LIN {X 0,Y 299.708,Z 457.98,A -85,B 0,C 180,E1 14084.743,E2 14084.743} C_VEL
LIN {X 0,Y 296.211,Z 453.711,A -85,B 0,C 180,E1 14082.616,E2 14082.616} C_VEL
LIN {X 0,Y 295.184,Z 452.077,A -85,B 0,C 180,E1 14081.599,E2 14081.599} C_VEL
LIN {X 0,Y 292.946,Z 448.012,A -85,B 0,C 180,E1 14078.654,E2 14078.654} C_VEL
LIN {X 0,Y 289.678,Z 442.411,A -85,B 0,C 180,E1 14073.523,E2 14073.523} C_VEL
LIN {X 0,Y 286.095,Z 436.55,A -85,B 0,C 180,E1 14064.796,E2 14064.796} C_VEL
LIN {X 0,Y 284.905,Z 435.389,A -85,B 0,C 180,E1 14059.25,E2 14059.25} C_VEL
LIN {X 0,Y 285.029,Z 435.504,A -85,B 0,C 180,E1 14053.387,E2 14053.387} C_VEL
LIN {X 0,Y 286.2,Z 436.707,A -85,B 0,C 180,E1 14048.438,E2 14048.438} C_VEL
LIN {X 0,Y 289.921,Z 442.675,A -85,B 0,C 180,E1 14039.803,E2 14039.803} C_VEL
LIN {X 0,Y 292.386,Z 447.018,A -85,B 0,C 180,E1 14035.882,E2 14035.882} C_VEL
LIN {X 0,Y 293.361,Z 448.287,A -85,B 0,C 180,E1 14034.721,E2 14034.721} C_VEL
LIN {X 0,Y 295.59,Z 452.337,A -85,B 0,C 180,E1 14031.833,E2 14031.833} C_VEL
LIN {X 0,Y 296.578,Z 453.696,A -85,B 0,C 180,E1 14030.884,E2 14030.884} C_VEL
LIN {X 0,Y 300.049,Z 458.18,A -85,B 0,C 180,E1 14028.662,E2 14028.662} C_VEL
LIN {X 0,Y 301.804,Z 460.211,A -85,B 0,C 180,E1 14027.662,E2 14027.662} C_VEL
LIN {X 0,Y 306.682,Z 466.167,A -85,B 0,C 180,E1 14025.124,E2 14025.124} C_VEL
LIN {X 0,Y 310.986,Z 471.496,A -85,B 0,C 180,E1 14023.085,E2 14023.085} C_VEL
LIN {X 0,Y 315.406,Z 477.154,A -85,B 0,C 180,E1 14021.135,E2 14021.135} C_VEL
LIN {X 0,Y 322.296,Z 486.098,A -85,B 0,C 180,E1 14018.384,E2 14018.384} C_VEL
LIN {X 0,Y 330.826,Z 498.047,A -85,B 0,C 180,E1 14015.303,E2 14015.303} C_VEL
LIN {X 0,Y 339.793,Z 511.207,A -85,B 0,C 180,E1 14012.39,E2 14012.39} C_VEL
LIN {X 0,Y 350.07,Z 527.48,A -85,B 0,C 180,E1 14009.372,E2 14009.372} C_VEL
LIN {X 0,Y 356.807,Z 539.249,A -85,B 0,C 180,E1 14007.536,E2 14007.536} C_VEL
LIN {X 0,Y 344.249,Z 751.792,A -85,B 0,C 180,E1 14003.107,E2 14003.107} C_VEL
LIN {X 0,Y 341.578,Z 773.987,A -85,B 0,C 180,E1 14002.425,E2 14002.425} C_VEL
LIN {X 0,Y 338.028,Z 795.147,A -85,B 0,C 180,E1 14001.526,E2 14001.526} C_VEL
LIN {X 0,Y 334.008,Z 814.782,A -85,B 0,C 180,E1 14000.432,E2 14000.432} C_VEL
LIN {X 0,Y 329.123,Z 834.708,A -85,B 0,C 180,E1 13999.01,E2 13999.01} C_VEL
LIN {X 0,Y 323.76,Z 853.792,A -85,B 0,C 180,E1 13997.311,E2 13997.311} C_VEL
LIN {X 0,Y 317.966,Z 872.343,A -85,B 0,C 180,E1 13995.293,E2 13995.293} C_VEL
LIN {X 0,Y 312.077,Z 889.799,A -85,B 0,C 180,E1 13992.972,E2 13992.972} C_VEL
LIN {X 0,Y 306.106,Z 906.312,A -85,B 0,C 180,E1 13990.3,E2 13990.3} C_VEL
LIN {X 0,Y 300.307,Z 921.84,A -85,B 0,C 180,E1 13987.276,E2 13987.276} C_VEL
LIN {X 0,Y 295.091,Z 935.845,A -85,B 0,C 180,E1 13983.995,E2 13983.995} C_VEL
LIN {X 0,Y 290.231,Z 949.123,A -85,B 0,C 180,E1 13980.201,E2 13980.201} C_VEL
LIN {X 0,Y 286.44,Z 960.225,A -85,B 0,C 180,E1 13976.319,E2 13976.319} C_VEL
LIN {X 0,Y 283.435,Z 970.371,A -85,B 0,C 180,E1 13971.962,E2 13971.962} C_VEL
LIN {X 0,Y 281.618,Z 978.164,A -85,B 0,C 180,E1 13967.782,E2 13967.782} C_VEL
LIN {X 0,Y 280.647,Z 984.135,A -85,B 0,C 180,E1 13963.604,E2 13963.604} C_VEL
LIN {X 0,Y 280.318,Z 988.504,A -85,B 0,C 180,E1 13959.448,E2 13959.448} C_VEL
LIN {X 0,Y 280.357,Z 991.092,A -85,B 0,C 180,E1 13955.727,E2 13955.727} C_VEL
LIN {X 0,Y 280.455,Z 992.448,A -85,B 0,C 180,E1 13951.843,E2 13951.843} C_VEL
LIN {X 0,Y 280.465,Z 992.441,A -85,B 0,C 180,E1 13948.37,E2 13948.37} C_VEL
LIN {X 0,Y 280.358,Z 991.198,A -85,B 0,C 180,E1 13944.479,E2 13944.479} C_VEL
LIN {X 0,Y 280.319,Z 988.431,A -85,B 0,C 180,E1 13940.561,E2 13940.561} C_VEL
LIN {X 0,Y 280.641,Z 984.136,A -85,B 0,C 180,E1 13936.405,E2 13936.405} C_VEL
LIN {X 0,Y 281.606,Z 978.138,A -85,B 0,C 180,E1 13932.226,E2 13932.226} C_VEL
LIN {X 0,Y 283.536,Z 970.074,A -85,B 0,C 180,E1 13927.837,E2 13927.837} C_VEL
LIN {X 0,Y 286.434,Z 960.623,A -85,B 0,C 180,E1 13923.69,E2 13923.69} C_VEL
LIN {X 0,Y 290.47,Z 949.125,A -85,B 0,C 180,E1 13919.608,E2 13919.608} C_VEL
LIN {X 0,Y 295.135,Z 936.858,A -85,B 0,C 180,E1 13916.02,E2 13916.02} C_VEL
LIN {X 0,Y 300.792,Z 922.545,A -85,B 0,C 180,E1 13912.539,E2 13912.539} C_VEL
LIN {X 0,Y 307.077,Z 906.789,A -85,B 0,C 180,E1 13909.374,E2 13909.374} C_VEL
LIN {X 0,Y 313.522,Z 889.976,A -85,B 0,C 180,E1 13906.607,E2 13906.607} C_VEL
LIN {X 0,Y 319.75,Z 872.82,A -85,B 0,C 180,E1 13904.275,E2 13904.275} C_VEL
LIN {X 0,Y 326.187,Z 853.924,A -85,B 0,C 180,E1 13902.167,E2 13902.167} C_VEL
LIN {X 0,Y 331.949,Z 835.118,A -85,B 0,C 180,E1 13900.459,E2 13900.459} C_VEL
LIN {X 0,Y 337.2,Z 815.456,A -85,B 0,C 180,E1 13899.032,E2 13899.032} C_VEL
LIN {X 0,Y 342.047,Z 794.262,A -85,B 0,C 180,E1 13897.824,E2 13897.824} C_VEL
LIN {X 0,Y 345.956,Z 773.376,A -85,B 0,C 180,E1 13896.928,E2 13896.928} C_VEL
LIN {X 0,Y 348.927,Z 751.08,A -85,B 0,C 180,E1 13896.239,E2 13896.239} C_VEL
LIN {X 0,Y 351.75,Z 711.318,A -85,B 0,C 180,E1 13895.359,E2 13895.359} C_VEL
LIN {X 0,Y 363.434,Z 540.393,A -85,B 0,C 180,E1 13891.741,E2 13891.741} C_VEL
LIN {X 0,Y 357.722,Z 529.548,A -85,B 0,C 180,E1 13889.559,E2 13889.559} C_VEL
LIN {X 0,Y 352.45,Z 520.256,A -85,B 0,C 180,E1 13887.268,E2 13887.268} C_VEL
LIN {X 0,Y 347.356,Z 511.98,A -85,B 0,C 180,E1 13884.669,E2 13884.669} C_VEL
LIN {X 0,Y 343.207,Z 505.565,A -85,B 0,C 180,E1 13882.074,E2 13882.074} C_VEL
LIN {X 0,Y 339.211,Z 499.557,A -85,B 0,C 180,E1 13878.74,E2 13878.74} C_VEL
LIN {X 0,Y 335.974,Z 494.822,A -85,B 0,C 180,E1 13873.948,E2 13873.948} C_VEL
LIN {X 0,Y 335.416,Z 494.331,A -85,B 0,C 180,E1 13869.956,E2 13869.956} C_VEL
LIN {X 0,Y 336.016,Z 495.136,A -85,B 0,C 180,E1 13867.695,E2 13867.695} C_VEL
LIN {X 0,Y 339.188,Z 499.976,A -85,B 0,C 180,E1 13863.041,E2 13863.041} C_VEL
LIN {X 0,Y 342.808,Z 505.592,A -85,B 0,C 180,E1 13859.954,E2 13859.954} C_VEL
LIN {X 0,Y 347.211,Z 512.447,A -85,B 0,C 180,E1 13857.148,E2 13857.148} C_VEL
LIN {X 0,Y 352.292,Z 520.969,A -85,B 0,C 180,E1 13854.503,E2 13854.503} C_VEL
LIN {X 0,Y 358.145,Z 531.437,A -85,B 0,C 180,E1 13851.935,E2 13851.935} C_VEL
LIN {X 0,Y 362.105,Z 539.53,A -85,B 0,C 180,E1 13850.361,E2 13850.361} C_VEL
LIN {X 0,Y 347.24,Z 729.778,A -85,B 0,C 180,E1 13846.162,E2 13846.162} C_VEL
LIN {X 0,Y 344.571,Z 750.475,A -85,B 0,C 180,E1 13845.442,E2 13845.442} C_VEL
LIN {X 0,Y 341.109,Z 770.29,A -85,B 0,C 180,E1 13844.496,E2 13844.496} C_VEL
LIN {X 0,Y 336.774,Z 790.108,A -85,B 0,C 180,E1 13843.262,E2 13843.262} C_VEL
LIN {X 0,Y 331.994,Z 808.511,A -85,B 0,C 180,E1 13841.821,E2 13841.821} C_VEL
LIN {X 0,Y 326.309,Z 827.229,A -85,B 0,C 180,E1 13839.985,E2 13839.985} C_VEL
LIN {X 0,Y 320.433,Z 844.262,A -85,B 0,C 180,E1 13837.917,E2 13837.917} C_VEL
LIN {X 0,Y 314.242,Z 860.65,A -85,B 0,C 180,E1 13835.492,E2 13835.492} C_VEL
LIN {X 0,Y 307.862,Z 876.286,A -85,B 0,C 180,E1 13832.643,E2 13832.643} C_VEL
LIN {X 0,Y 301.914,Z 890.087,A -85,B 0,C 180,E1 13829.555,E2 13829.555} C_VEL
LIN {X 0,Y 296.711,Z 901.883,A -85,B 0,C 180,E1 13826.33,E2 13826.33} C_VEL
LIN {X 0,Y 291.707,Z 913.109,A -85,B 0,C 180,E1 13822.51,E2 13822.51} C_VEL
LIN {X 0,Y 287.771,Z 922.132,A -85,B 0,C 180,E1 13818.624,E2 13818.624} C_VEL
LIN {X 0,Y 284.793,Z 929.43,A -85,B 0,C 180,E1 13814.593,E2 13814.593} C_VEL
LIN {X 0,Y 282.677,Z 935.212,A -85,B 0,C 180,E1 13810.33,E2 13810.33} C_VEL
LIN {X 0,Y 281.469,Z 939.176,A -85,B 0,C 180,E1 13806.128,E2 13806.128} C_VEL
LIN {X 0,Y 280.884,Z 941.516,A -85,B 0,C 180,E1 13802.026,E2 13802.026} C_VEL
LIN {X 0,Y 280.668,Z 942.269,A -85,B 0,C 180,E1 13798.044,E2 13798.044} C_VEL
LIN {X 0,Y 280.694,Z 941.642,A -85,B 0,C 180,E1 13793.953,E2 13793.953} C_VEL
LIN {X 0,Y 281.006,Z 939.657,A -85,B 0,C 180,E1 13789.968,E2 13789.968} C_VEL
LIN {X 0,Y 281.746,Z 936.002,A -85,B 0,C 180,E1 13785.853,E2 13785.853} C_VEL
LIN {X 0,Y 283.125,Z 930.815,A -85,B 0,C 180,E1 13781.815,E2 13781.815} C_VEL
LIN {X 0,Y 285.464,Z 923.534,A -85,B 0,C 180,E1 13777.589,E2 13777.589} C_VEL
LIN {X 0,Y 288.566,Z 914.907,A -85,B 0,C 180,E1 13773.707,E2 13773.707} C_VEL
LIN {X 0,Y 292.502,Z 904.595,A -85,B 0,C 180,E1 13769.996,E2 13769.996} C_VEL
LIN {X 0,Y 297.15,Z 892.639,A -85,B 0,C 180,E1 13766.524,E2 13766.524} C_VEL
LIN {X 0,Y 302.287,Z 879.189,A -85,B 0,C 180,E1 13763.348,E2 13763.348} C_VEL
LIN {X 0,Y 307.603,Z 864.78,A -85,B 0,C 180,E1 13760.552,E2 13760.552} C_VEL
LIN {X 0,Y 313.308,Z 848.33,A -85,B 0,C 180,E1 13757.931,E2 13757.931} C_VEL
LIN {X 0,Y 318.871,Z 830.822,A -85,B 0,C 180,E1 13755.654,E2 13755.654} C_VEL
LIN {X 0,Y 323.952,Z 813.125,A -85,B 0,C 180,E1 13753.777,E2 13753.777} C_VEL
LIN {X 0,Y 328.802,Z 793.678,A -85,B 0,C 180,E1 13752.11,E2 13752.11} C_VEL
LIN {X 0,Y 332.844,Z 774.169,A -85,B 0,C 180,E1 13750.793,E2 13750.793} C_VEL
LIN {X 0,Y 336.296,Z 753.654,A -85,B 0,C 180,E1 13749.726,E2 13749.726} C_VEL
LIN {X 0,Y 339.018,Z 732.049,A -85,B 0,C 180,E1 13748.908,E2 13748.908} C_VEL
LIN {X 0,Y 341.02,Z 706.482,A -85,B 0,C 180,E1 13748.266,E2 13748.266} C_VEL
LIN {X 0,Y 346.591,Z 617.799,A -85,B 0,C 180,E1 13746.355,E2 13746.355} C_VEL
LIN {X 0,Y 346.441,Z 610.234,A -85,B 0,C 180,E1 13746.064,E2 13746.064} C_VEL
LIN {X 0,Y 343.807,Z 590.496,A -85,B 0,C 180,E1 13744.832,E2 13744.832} C_VEL
LIN {X 0,Y 343.792,Z 583.99,A -85,B 0,C 180,E1 13744.597,E2 13744.597} C_VEL
LIN {X 0,Y 346.817,Z 537.187,A -85,B 0,C 180,E1 13743.577,E2 13743.577} C_VEL
LIN {X 0,Y 337.141,Z 520.499,A -85,B 0,C 180,E1 13740.683,E2 13740.683} C_VEL
LIN {X 0,Y 328.675,Z 507.267,A -85,B 0,C 180,E1 13737.912,E2 13737.912} C_VEL
LIN {X 0,Y 320.316,Z 494.892,A -85,B 0,C 180,E1 13734.869,E2 13734.869} C_VEL
LIN {X 0,Y 313.183,Z 485.205,A -85,B 0,C 180,E1 13731.985,E2 13731.985} C_VEL
LIN {X 0,Y 309.567,Z 480.371,A -85,B 0,C 180,E1 13730.384,E2 13730.384} C_VEL
LIN {X 0,Y 304.803,Z 474.227,A -85,B 0,C 180,E1 13728.129,E2 13728.129} C_VEL
LIN {X 0,Y 301.44,Z 470.025,A -85,B 0,C 180,E1 13726.372,E2 13726.372} C_VEL
LIN {X 0,Y 297.75,Z 465.415,A -85,B 0,C 180,E1 13724.305,E2 13724.305} C_VEL
LIN {X 0,Y 293.97,Z 460.61,A -85,B 0,C 180,E1 13721.94,E2 13721.94} C_VEL
LIN {X 0,Y 289.516,Z 455.7,A -85,B 0,C 180,E1 13718.817,E2 13718.817} C_VEL
LIN {X 0,Y 288.116,Z 453.799,A -85,B 0,C 180,E1 13717.647,E2 13717.647} C_VEL
LIN {X 0,Y 285.424,Z 449.327,A -85,B 0,C 180,E1 13713.511,E2 13713.511} C_VEL
LIN {X 0,Y 283.51,Z 446.932,A -85,B 0,C 180,E1 13710.053,E2 13710.053} C_VEL
LIN {X 0,Y 281.927,Z 443.33,A -85,B 0,C 180,E1 13704.516,E2 13704.516} C_VEL
LIN {X 0,Y 280.804,Z 442.247,A -85,B 0,C 180,E1 13698.692,E2 13698.692} C_VEL
LIN {X 0,Y 281.057,Z 442.483,A -85,B 0,C 180,E1 13692.952,E2 13692.952} C_VEL
LIN {X 0,Y 282.155,Z 443.658,A -85,B 0,C 180,E1 13688.355,E2 13688.355} C_VEL
LIN {X 0,Y 285.729,Z 449.423,A -85,B 0,C 180,E1 13680.001,E2 13680.001} C_VEL
LIN {X 0,Y 288.198,Z 453.801,A -85,B 0,C 180,E1 13676.022,E2 13676.022} C_VEL
LIN {X 0,Y 289.577,Z 455.388,A -85,B 0,C 180,E1 13674.85,E2 13674.85} C_VEL
LIN {X 0,Y 293.081,Z 459.681,A -85,B 0,C 180,E1 13672.256,E2 13672.256} C_VEL
LIN {X 0,Y 294.815,Z 461.548,A -85,B 0,C 180,E1 13671.124,E2 13671.124} C_VEL
LIN {X 0,Y 298.661,Z 466.098,A -85,B 0,C 180,E1 13668.804,E2 13668.804} C_VEL
LIN {X 0,Y 304.61,Z 473.584,A -85,B 0,C 180,E1 13665.547,E2 13665.547} C_VEL
LIN {X 0,Y 308.777,Z 478.808,A -85,B 0,C 180,E1 13663.541,E2 13663.541} C_VEL
LIN {X 0,Y 313.027,Z 484.349,A -85,B 0,C 180,E1 13661.614,E2 13661.614} C_VEL
LIN {X 0,Y 319.731,Z 493.188,A -85,B 0,C 180,E1 13658.875,E2 13658.875} C_VEL
LIN {X 0,Y 329.277,Z 506.679,A -85,B 0,C 180,E1 13655.37,E2 13655.37} C_VEL
LIN {X 0,Y 339.871,Z 522.854,A -85,B 0,C 180,E1 13651.921,E2 13651.921} C_VEL
LIN {X 0,Y 350.632,Z 540.799,A -85,B 0,C 180,E1 13648.784,E2 13648.784} C_VEL
LIN {X 0,Y 351.67,Z 542.991,A -85,B 0,C 180,E1 13648.484,E2 13648.484} C_VEL
LIN {X 0,Y 338.923,Z 751.325,A -85,B 0,C 180,E1 13644.117,E2 13644.117} C_VEL
LIN {X 0,Y 336.179,Z 773.519,A -85,B 0,C 180,E1 13643.433,E2 13643.433} C_VEL
LIN {X 0,Y 332.556,Z 794.521,A -85,B 0,C 180,E1 13642.54,E2 13642.54} C_VEL
LIN {X 0,Y 328.218,Z 814.967,A -85,B 0,C 180,E1 13641.391,E2 13641.391} C_VEL
LIN {X 0,Y 323.11,Z 835.108,A -85,B 0,C 180,E1 13639.936,E2 13639.936} C_VEL
LIN {X 0,Y 317.653,Z 853.772,A -85,B 0,C 180,E1 13638.248,E2 13638.248} C_VEL
LIN {X 0,Y 311.419,Z 872.942,A -85,B 0,C 180,E1 13636.124,E2 13636.124} C_VEL
LIN {X 0,Y 305.233,Z 890.589,A -85,B 0,C 180,E1 13633.727,E2 13633.727} C_VEL
LIN {X 0,Y 299.16,Z 906.676,A -85,B 0,C 180,E1 13631.056,E2 13631.056} C_VEL
LIN {X 0,Y 293.007,Z 922.387,A -85,B 0,C 180,E1 13627.9,E2 13627.9} C_VEL
LIN {X 0,Y 287.532,Z 936.372,A -85,B 0,C 180,E1 13624.5,E2 13624.5} C_VEL
LIN {X 0,Y 282.639,Z 949.192,A -85,B 0,C 180,E1 13620.726,E2 13620.726} C_VEL
LIN {X 0,Y 278.613,Z 960.398,A -85,B 0,C 180,E1 13616.657,E2 13616.657} C_VEL
LIN {X 0,Y 275.625,Z 969.939,A -85,B 0,C 180,E1 13612.393,E2 13612.393} C_VEL
LIN {X 0,Y 273.704,Z 977.669,A -85,B 0,C 180,E1 13608.094,E2 13608.094} C_VEL
LIN {X 0,Y 272.681,Z 983.613,A -85,B 0,C 180,E1 13603.793,E2 13603.793} C_VEL
LIN {X 0,Y 272.336,Z 987.917,A -85,B 0,C 180,E1 13599.514,E2 13599.514} C_VEL
LIN {X 0,Y 272.383,Z 990.465,A -85,B 0,C 180,E1 13595.692,E2 13595.692} C_VEL
LIN {X 0,Y 272.491,Z 991.749,A -85,B 0,C 180,E1 13591.687,E2 13591.687} C_VEL
LIN {X 0,Y 272.488,Z 991.694,A -85,B 0,C 180,E1 13588.112,E2 13588.112} C_VEL
LIN {X 0,Y 272.377,Z 990.371,A -85,B 0,C 180,E1 13584.105,E2 13584.105} C_VEL
LIN {X 0,Y 272.344,Z 987.545,A -85,B 0,C 180,E1 13580.069,E2 13580.069} C_VEL
LIN {X 0,Y 272.739,Z 983.152,A -85,B 0,C 180,E1 13575.787,E2 13575.787} C_VEL
LIN {X 0,Y 273.832,Z 977.096,A -85,B 0,C 180,E1 13571.483,E2 13571.483} C_VEL
LIN {X 0,Y 276.004,Z 968.894,A -85,B 0,C 180,E1 13566.946,E2 13566.946} C_VEL
LIN {X 0,Y 279.25,Z 959.124,A -85,B 0,C 180,E1 13562.618,E2 13562.618} C_VEL
LIN {X 0,Y 283.534,Z 947.851,A -85,B 0,C 180,E1 13558.546,E2 13558.546} C_VEL
LIN {X 0,Y 288.631,Z 935.27,A -85,B 0,C 180,E1 13554.838,E2 13554.838} C_VEL
LIN {X 0,Y 294.731,Z 920.709,A -85,B 0,C 180,E1 13551.284,E2 13551.284} C_VEL
LIN {X 0,Y 301.02,Z 905.688,A -85,B 0,C 180,E1 13548.25,E2 13548.25} C_VEL
LIN {X 0,Y 308.05,Z 888.24,A -85,B 0,C 180,E1 13545.363,E2 13545.363} C_VEL
LIN {X 0,Y 314.572,Z 870.988,A -85,B 0,C 180,E1 13543.033,E2 13543.033} C_VEL
LIN {X 0,Y 321.378,Z 851.578,A -85,B 0,C 180,E1 13540.894,E2 13540.894} C_VEL
LIN {X 0,Y 327.267,Z 833.033,A -85,B 0,C 180,E1 13539.228,E2 13539.228} C_VEL
LIN {X 0,Y 332.755,Z 812.973,A -85,B 0,C 180,E1 13537.799,E2 13537.799} C_VEL
LIN {X 0,Y 337.626,Z 791.945,A -85,B 0,C 180,E1 13536.634,E2 13536.634} C_VEL
LIN {X 0,Y 341.701,Z 770.294,A -85,B 0,C 180,E1 13535.74,E2 13535.74} C_VEL
LIN {X 0,Y 344.659,Z 748.232,A -85,B 0,C 180,E1 13535.075,E2 13535.075} C_VEL
LIN {X 0,Y 359.241,Z 544.487,A -85,B 0,C 180,E1 13530.712,E2 13530.712} C_VEL
LIN {X 0,Y 354.267,Z 534.778,A -85,B 0,C 180,E1 13528.672,E2 13528.672} C_VEL
LIN {X 0,Y 349.671,Z 526.511,A -85,B 0,C 180,E1 13526.537,E2 13526.537} C_VEL
LIN {X 0,Y 345.053,Z 518.755,A -85,B 0,C 180,E1 13524.024,E2 13524.024} C_VEL
LIN {X 0,Y 340.926,Z 512.002,A -85,B 0,C 180,E1 13521.235,E2 13521.235} C_VEL
LIN {X 0,Y 337.668,Z 507.121,A -85,B 0,C 180,E1 13518.292,E2 13518.292} C_VEL
LIN {X 0,Y 334.843,Z 502.711,A -85,B 0,C 180,E1 13513.82,E2 13513.82} C_VEL
LIN {X 0,Y 334.357,Z 502.266,A -85,B 0,C 180,E1 13509.814,E2 13509.814} C_VEL
LIN {X 0,Y 334.923,Z 503.164,A -85,B 0,C 180,E1 13507.676,E2 13507.676} C_VEL
LIN {X 0,Y 337.799,Z 507.725,A -85,B 0,C 180,E1 13503.308,E2 13503.308} C_VEL
LIN {X 0,Y 341.134,Z 513.076,A -85,B 0,C 180,E1 13500.335,E2 13500.335} C_VEL
LIN {X 0,Y 345.225,Z 519.754,A -85,B 0,C 180,E1 13497.587,E2 13497.587} C_VEL
LIN {X 0,Y 350.054,Z 528.14,A -85,B 0,C 180,E1 13494.961,E2 13494.961} C_VEL
LIN {X 0,Y 355.603,Z 538.509,A -85,B 0,C 180,E1 13492.406,E2 13492.406} C_VEL
LIN {X 0,Y 357.996,Z 543.629,A -85,B 0,C 180,E1 13491.401,E2 13491.401} C_VEL
LIN {X 0,Y 342.803,Z 730.135,A -85,B 0,C 180,E1 13487.267,E2 13487.267} C_VEL
LIN {X 0,Y 340.028,Z 750.857,A -85,B 0,C 180,E1 13486.546,E2 13486.546} C_VEL
LIN {X 0,Y 336.315,Z 771.352,A -85,B 0,C 180,E1 13485.564,E2 13485.564} C_VEL
LIN {X 0,Y 331.742,Z 791.394,A -85,B 0,C 180,E1 13484.305,E2 13484.305} C_VEL
LIN {X 0,Y 326.542,Z 810.369,A -85,B 0,C 180,E1 13482.792,E2 13482.792} C_VEL
LIN {X 0,Y 320.554,Z 829.191,A -85,B 0,C 180,E1 13480.91,E2 13480.91} C_VEL
LIN {X 0,Y 314.283,Z 846.549,A -85,B 0,C 180,E1 13478.757,E2 13478.757} C_VEL
LIN {X 0,Y 308.149,Z 861.893,A -85,B 0,C 180,E1 13476.425,E2 13476.425} C_VEL
LIN {X 0,Y 301.5,Z 877.401,A -85,B 0,C 180,E1 13473.547,E2 13473.547} C_VEL
LIN {X 0,Y 295.173,Z 891.325,A -85,B 0,C 180,E1 13470.359,E2 13470.359} C_VEL
LIN {X 0,Y 289.485,Z 903.468,A -85,B 0,C 180,E1 13466.926,E2 13466.926} C_VEL
LIN {X 0,Y 284.527,Z 914.01,A -85,B 0,C 180,E1 13463.237,E2 13463.237} C_VEL
LIN {X 0,Y 280.239,Z 923.241,A -85,B 0,C 180,E1 13459.138,E2 13459.138} C_VEL
LIN {X 0,Y 277.076,Z 930.474,A -85,B 0,C 180,E1 13454.984,E2 13454.984} C_VEL
LIN {X 0,Y 274.84,Z 936.137,A -85,B 0,C 180,E1 13450.624,E2 13450.624} C_VEL
LIN {X 0,Y 273.493,Z 940.185,A -85,B 0,C 180,E1 13446.051,E2 13446.051} C_VEL
LIN {X 0,Y 272.9,Z 942.371,A -85,B 0,C 180,E1 13441.786,E2 13441.786} C_VEL
LIN {X 0,Y 272.695,Z 943.015,A -85,B 0,C 180,E1 13437.747,E2 13437.747} C_VEL
LIN {X 0,Y 272.74,Z 942.231,A -85,B 0,C 180,E1 13433.547,E2 13433.547} C_VEL
LIN {X 0,Y 273.133,Z 939.921,A -85,B 0,C 180,E1 13429.231,E2 13429.231} C_VEL
LIN {X 0,Y 274.014,Z 936.131,A -85,B 0,C 180,E1 13425.01,E2 13425.01} C_VEL
LIN {X 0,Y 275.711,Z 930.395,A -85,B 0,C 180,E1 13420.647,E2 13420.647} C_VEL
LIN {X 0,Y 278.164,Z 923.29,A -85,B 0,C 180,E1 13416.6,E2 13416.6} C_VEL
LIN {X 0,Y 281.547,Z 914.445,A -85,B 0,C 180,E1 13412.642,E2 13412.642} C_VEL
LIN {X 0,Y 285.632,Z 904.301,A -85,B 0,C 180,E1 13408.993,E2 13408.993} C_VEL
LIN {X 0,Y 290.298,Z 892.919,A -85,B 0,C 180,E1 13405.65,E2 13405.65} C_VEL
LIN {X 0,Y 295.693,Z 879.382,A -85,B 0,C 180,E1 13402.418,E2 13402.418} C_VEL
LIN {X 0,Y 301.273,Z 864.846,A -85,B 0,C 180,E1 13399.576,E2 13399.576} C_VEL
LIN {X 0,Y 307.011,Z 848.908,A -85,B 0,C 180,E1 13397.01,E2 13397.01} C_VEL
LIN {X 0,Y 312.794,Z 831.387,A -85,B 0,C 180,E1 13394.706,E2 13394.706} C_VEL
LIN {X 0,Y 318.061,Z 813.685,A -85,B 0,C 180,E1 13392.809,E2 13392.809} C_VEL
LIN {X 0,Y 323.082,Z 794.232,A -85,B 0,C 180,E1 13391.128,E2 13391.128} C_VEL
LIN {X 0,Y 327.265,Z 774.725,A -85,B 0,C 180,E1 13389.8,E2 13389.8} C_VEL
LIN {X 0,Y 330.831,Z 754.216,A -85,B 0,C 180,E1 13388.727,E2 13388.727} C_VEL
LIN {X 0,Y 333.657,Z 732.507,A -85,B 0,C 180,E1 13387.9,E2 13387.9} C_VEL
LIN {X 0,Y 335.728,Z 706.989,A -85,B 0,C 180,E1 13387.253,E2 13387.253} C_VEL
LIN {X 0,Y 343.792,Z 583.99,A -85,B 0,C 180,E1 13384.597,E2 13384.597} C_VEL
LIN {X 0,Y 343.707,Z 576.423,A -85,B 0,C 180,E1 13384.308,E2 13384.308} C_VEL
LIN {X 0,Y 341.288,Z 556.687,A -85,B 0,C 180,E1 13383.052,E2 13383.052} C_VEL
LIN {X 0,Y 341.286,Z 550.183,A -85,B 0,C 180,E1 13382.81,E2 13382.81} C_VEL
LIN {X 0,Y 341.857,Z 540.878,A -85,B 0,C 180,E1 13382.592,E2 13382.592} C_VEL
LIN {X 0,Y 332.474,Z 524.8,A -85,B 0,C 180,E1 13379.668,E2 13379.668} C_VEL
LIN {X 0,Y 324.131,Z 511.493,A -85,B 0,C 180,E1 13376.798,E2 13376.798} C_VEL
LIN {X 0,Y 314.969,Z 498.115,A -85,B 0,C 180,E1 13373.28,E2 13373.28} C_VEL
LIN {X 0,Y 307.65,Z 488.044,A -85,B 0,C 180,E1 13370.086,E2 13370.086} C_VEL
LIN {X 0,Y 300.681,Z 478.781,A -85,B 0,C 180,E1 13366.601,E2 13366.601} C_VEL
LIN {X 0,Y 295.635,Z 472.68,A -85,B 0,C 180,E1 13363.76,E2 13363.76} C_VEL
LIN {X 0,Y 291.404,Z 467.296,A -85,B 0,C 180,E1 13360.983,E2 13360.983} C_VEL
LIN {X 0,Y 287.692,Z 463.012,A -85,B 0,C 180,E1 13358.28,E2 13358.28} C_VEL
LIN {X 0,Y 286.341,Z 461.31,A -85,B 0,C 180,E1 13357.164,E2 13357.164} C_VEL
LIN {X 0,Y 282.442,Z 456.938,A -85,B 0,C 180,E1 13353.522,E2 13353.522} C_VEL
LIN {X 0,Y 281.057,Z 455.343,A -85,B 0,C 180,E1 13352.011,E2 13352.011} C_VEL
LIN {X 0,Y 278.183,Z 451.331,A -85,B 0,C 180,E1 13346.468,E2 13346.468} C_VEL
LIN {X 0,Y 277.643,Z 450.006,A -85,B 0,C 180,E1 13343.788,E2 13343.788} C_VEL
LIN {X 0,Y 276.711,Z 449.119,A -85,B 0,C 180,E1 13337.887,E2 13337.887} C_VEL
LIN {X 0,Y 277.126,Z 449.511,A -85,B 0,C 180,E1 13332.291,E2 13332.291} C_VEL
LIN {X 0,Y 278.092,Z 450.642,A -85,B 0,C 180,E1 13328.269,E2 13328.269} C_VEL
LIN {X 0,Y 281.509,Z 455.696,A -85,B 0,C 180,E1 13321.222,E2 13321.222} C_VEL
LIN {X 0,Y 282.867,Z 457.267,A -85,B 0,C 180,E1 13319.798,E2 13319.798} C_VEL
LIN {X 0,Y 287.095,Z 461.929,A -85,B 0,C 180,E1 13315.906,E2 13315.906} C_VEL
LIN {X 0,Y 291.578,Z 467.432,A -85,B 0,C 180,E1 13312.513,E2 13312.513} C_VEL
LIN {X 0,Y 293.128,Z 469.238,A -85,B 0,C 180,E1 13311.468,E2 13311.468} C_VEL
LIN {X 0,Y 297.097,Z 473.866,A -85,B 0,C 180,E1 13309.039,E2 13309.039} C_VEL
LIN {X 0,Y 305.59,Z 484.627,A -85,B 0,C 180,E1 13304.486,E2 13304.486} C_VEL
LIN {X 0,Y 311.531,Z 492.736,A -85,B 0,C 180,E1 13301.717,E2 13301.717} C_VEL
LIN {X 0,Y 317.363,Z 500.568,A -85,B 0,C 180,E1 13299.29,E2 13299.29} C_VEL
LIN {X 0,Y 326.361,Z 513.502,A -85,B 0,C 180,E1 13295.907,E2 13295.907} C_VEL
LIN {X 0,Y 336.536,Z 529.258,A -85,B 0,C 180,E1 13292.509,E2 13292.509} C_VEL
LIN {X 0,Y 346.644,Z 546.37,A -85,B 0,C 180,E1 13289.469,E2 13289.469} C_VEL
LIN {X 0,Y 333.637,Z 751.083,A -85,B 0,C 180,E1 13285.146,E2 13285.146} C_VEL
LIN {X 0,Y 330.802,Z 773.371,A -85,B 0,C 180,E1 13284.455,E2 13284.455} C_VEL
LIN {X 0,Y 326.983,Z 794.787,A -85,B 0,C 180,E1 13283.538,E2 13283.538} C_VEL
LIN {X 0,Y 322.325,Z 815.873,A -85,B 0,C 180,E1 13282.332,E2 13282.332} C_VEL
LIN {X 0,Y 317.094,Z 835.828,A -85,B 0,C 180,E1 13280.871,E2 13280.871} C_VEL
LIN {X 0,Y 311.367,Z 854.587,A -85,B 0,C 180,E1 13279.137,E2 13279.137} C_VEL
LIN {X 0,Y 304.939,Z 873.516,A -85,B 0,C 180,E1 13276.99,E2 13276.99} C_VEL
LIN {X 0,Y 298.545,Z 890.968,A -85,B 0,C 180,E1 13274.562,E2 13274.562} C_VEL
LIN {X 0,Y 291.965,Z 907.759,A -85,B 0,C 180,E1 13271.708,E2 13271.708} C_VEL
LIN {X 0,Y 285.704,Z 923.016,A -85,B 0,C 180,E1 13268.535,E2 13268.535} C_VEL
LIN {X 0,Y 279.773,Z 937.432,A -85,B 0,C 180,E1 13264.881,E2 13264.881} C_VEL
LIN {X 0,Y 274.866,Z 949.685,A -85,B 0,C 180,E1 13261.105,E2 13261.105} C_VEL
LIN {X 0,Y 270.797,Z 960.545,A -85,B 0,C 180,E1 13257.014,E2 13257.014} C_VEL
LIN {X 0,Y 267.76,Z 969.73,A -85,B 0,C 180,E1 13252.731,E2 13252.731} C_VEL
LIN {X 0,Y 265.722,Z 977.495,A -85,B 0,C 180,E1 13248.203,E2 13248.203} C_VEL
LIN {X 0,Y 264.68,Z 983.353,A -85,B 0,C 180,E1 13243.772,E2 13243.772} C_VEL
LIN {X 0,Y 264.353,Z 987.495,A -85,B 0,C 180,E1 13239.364,E2 13239.364} C_VEL
LIN {X 0,Y 264.415,Z 990.066,A -85,B 0,C 180,E1 13235.211,E2 13235.211} C_VEL
LIN {X 0,Y 264.531,Z 991.069,A -85,B 0,C 180,E1 13231.304,E2 13231.304} C_VEL
LIN {X 0,Y 264.501,Z 990.914,A -85,B 0,C 180,E1 13227.622,E2 13227.622} C_VEL
LIN {X 0,Y 264.386,Z 989.407,A -85,B 0,C 180,E1 13223.49,E2 13223.49} C_VEL
LIN {X 0,Y 264.385,Z 986.618,A -85,B 0,C 180,E1 13219.504,E2 13219.504} C_VEL
LIN {X 0,Y 264.884,Z 981.892,A -85,B 0,C 180,E1 13214.908,E2 13214.908} C_VEL
LIN {X 0,Y 266.181,Z 975.733,A -85,B 0,C 180,E1 13210.475,E2 13210.475} C_VEL
LIN {X 0,Y 268.497,Z 967.817,A -85,B 0,C 180,E1 13206.058,E2 13206.058} C_VEL
LIN {X 0,Y 272.183,Z 957.633,A -85,B 0,C 180,E1 13201.48,E2 13201.48} C_VEL
LIN {X 0,Y 276.914,Z 946.087,A -85,B 0,C 180,E1 13197.276,E2 13197.276} C_VEL
LIN {X 0,Y 282.478,Z 933.226,A -85,B 0,C 180,E1 13193.464,E2 13193.464} C_VEL
LIN {X 0,Y 288.513,Z 919.585,A -85,B 0,C 180,E1 13190.131,E2 13190.131} C_VEL
LIN {X 0,Y 295.265,Z 904.218,A -85,B 0,C 180,E1 13187.007,E2 13187.007} C_VEL
LIN {X 0,Y 302.189,Z 887.836,A -85,B 0,C 180,E1 13184.277,E2 13184.277} C_VEL
LIN {X 0,Y 309.031,Z 870.566,A -85,B 0,C 180,E1 13181.921,E2 13181.921} C_VEL
LIN {X 0,Y 316.091,Z 851.262,A -85,B 0,C 180,E1 13179.775,E2 13179.775} C_VEL
LIN {X 0,Y 322.437,Z 831.93,A -85,B 0,C 180,E1 13178.043,E2 13178.043} C_VEL
LIN {X 0,Y 328.177,Z 811.727,A -85,B 0,C 180,E1 13176.61,E2 13176.61} C_VEL
LIN {X 0,Y 333.058,Z 791.344,A -85,B 0,C 180,E1 13175.49,E2 13175.49} C_VEL
LIN {X 0,Y 337.299,Z 769.439,A -85,B 0,C 180,E1 13174.595,E2 13174.595} C_VEL
LIN {X 0,Y 340.32,Z 747.358,A -85,B 0,C 180,E1 13173.934,E2 13173.934} C_VEL
LIN {X 0,Y 355.224,Z 548.583,A -85,B 0,C 180,E1 13169.649,E2 13169.649} C_VEL
LIN {X 0,Y 350.367,Z 538.956,A -85,B 0,C 180,E1 13167.489,E2 13167.489} C_VEL
LIN {X 0,Y 345.72,Z 530.495,A -85,B 0,C 180,E1 13165.113,E2 13165.113} C_VEL
LIN {X 0,Y 341.582,Z 523.311,A -85,B 0,C 180,E1 13162.547,E2 13162.547} C_VEL
LIN {X 0,Y 338.722,Z 518.798,A -85,B 0,C 180,E1 13160.384,E2 13160.384} C_VEL
LIN {X 0,Y 336.306,Z 514.851,A -85,B 0,C 180,E1 13158.01,E2 13158.01} C_VEL
LIN {X 0,Y 333.714,Z 510.601,A -85,B 0,C 180,E1 13153.691,E2 13153.691} C_VEL
LIN {X 0,Y 333.299,Z 510.211,A -85,B 0,C 180,E1 13149.671,E2 13149.671} C_VEL
LIN {X 0,Y 333.798,Z 511.112,A -85,B 0,C 180,E1 13147.746,E2 13147.746} C_VEL
LIN {X 0,Y 336.418,Z 515.473,A -85,B 0,C 180,E1 13143.578,E2 13143.578} C_VEL
LIN {X 0,Y 339.635,Z 520.856,A -85,B 0,C 180,E1 13140.59,E2 13140.59} C_VEL
LIN {X 0,Y 343.439,Z 527.417,A -85,B 0,C 180,E1 13137.914,E2 13137.914} C_VEL
LIN {X 0,Y 347.917,Z 535.449,A -85,B 0,C 180,E1 13135.384,E2 13135.384} C_VEL
LIN {X 0,Y 353.297,Z 545.949,A -85,B 0,C 180,E1 13132.805,E2 13132.805} C_VEL
LIN {X 0,Y 354.021,Z 547.837,A -85,B 0,C 180,E1 13132.463,E2 13132.463} C_VEL
LIN {X 0,Y 338.513,Z 730.77,A -85,B 0,C 180,E1 13128.398,E2 13128.398} C_VEL
LIN {X 0,Y 335.653,Z 751.425,A -85,B 0,C 180,E1 13127.679,E2 13127.679} C_VEL
LIN {X 0,Y 331.819,Z 771.81,A -85,B 0,C 180,E1 13126.702,E2 13126.702} C_VEL
LIN {X 0,Y 326.998,Z 792.104,A -85,B 0,C 180,E1 13125.424,E2 13125.424} C_VEL
LIN {X 0,Y 321.547,Z 811.21,A -85,B 0,C 180,E1 13123.893,E2 13123.893} C_VEL
LIN {X 0,Y 315.343,Z 829.954,A -85,B 0,C 180,E1 13122.01,E2 13122.01} C_VEL
LIN {X 0,Y 308.826,Z 847.204,A -85,B 0,C 180,E1 13119.852,E2 13119.852} C_VEL
LIN {X 0,Y 302.147,Z 863.202,A -85,B 0,C 180,E1 13117.392,E2 13117.392} C_VEL
LIN {X 0,Y 295.323,Z 878.335,A -85,B 0,C 180,E1 13114.533,E2 13114.533} C_VEL
LIN {X 0,Y 288.499,Z 892.578,A -85,B 0,C 180,E1 13111.201,E2 13111.201} C_VEL
LIN {X 0,Y 282.526,Z 904.643,A -85,B 0,C 180,E1 13107.697,E2 13107.697} C_VEL
LIN {X 0,Y 277.418,Z 914.862,A -85,B 0,C 180,E1 13104.021,E2 13104.021} C_VEL
LIN {X 0,Y 272.732,Z 924.371,A -85,B 0,C 180,E1 13099.68,E2 13099.68} C_VEL
LIN {X 0,Y 269.398,Z 931.464,A -85,B 0,C 180,E1 13095.438,E2 13095.438} C_VEL
LIN {X 0,Y 267.12,Z 936.782,A -85,B 0,C 180,E1 13091.2,E2 13091.2} C_VEL
LIN {X 0,Y 265.689,Z 940.716,A -85,B 0,C 180,E1 13086.718,E2 13086.718} C_VEL
LIN {X 0,Y 264.985,Z 943.027,A -85,B 0,C 180,E1 13082.304,E2 13082.304} C_VEL
LIN {X 0,Y 264.735,Z 943.719,A -85,B 0,C 180,E1 13078.165,E2 13078.165} C_VEL
LIN {X 0,Y 264.763,Z 943.058,A -85,B 0,C 180,E1 13073.827,E2 13073.827} C_VEL
LIN {X 0,Y 265.123,Z 941.048,A -85,B 0,C 180,E1 13069.606,E2 13069.606} C_VEL
LIN {X 0,Y 265.977,Z 937.376,A -85,B 0,C 180,E1 13065.251,E2 13065.251} C_VEL
LIN {X 0,Y 267.563,Z 932.17,A -85,B 0,C 180,E1 13060.982,E2 13060.982} C_VEL
LIN {X 0,Y 270.172,Z 924.978,A -85,B 0,C 180,E1 13056.583,E2 13056.583} C_VEL
LIN {X 0,Y 273.627,Z 916.383,A -85,B 0,C 180,E1 13052.509,E2 13052.509} C_VEL
LIN {X 0,Y 277.812,Z 906.5,A -85,B 0,C 180,E1 13048.758,E2 13048.758} C_VEL
LIN {X 0,Y 283.022,Z 894.278,A -85,B 0,C 180,E1 13045.043,E2 13045.043} C_VEL
LIN {X 0,Y 288.467,Z 881.242,A -85,B 0,C 180,E1 13041.826,E2 13041.826} C_VEL
LIN {X 0,Y 294.428,Z 866.435,A -85,B 0,C 180,E1 13038.835,E2 13038.835} C_VEL
LIN {X 0,Y 300.582,Z 850.075,A -85,B 0,C 180,E1 13036.139,E2 13036.139} C_VEL
LIN {X 0,Y 306.345,Z 833.365,A -85,B 0,C 180,E1 13033.89,E2 13033.89} C_VEL
LIN {X 0,Y 312.021,Z 815.064,A -85,B 0,C 180,E1 13031.887,E2 13031.887} C_VEL
LIN {X 0,Y 317.196,Z 795.688,A -85,B 0,C 180,E1 13030.189,E2 13030.189} C_VEL
LIN {X 0,Y 321.514,Z 776.409,A -85,B 0,C 180,E1 13028.851,E2 13028.851} C_VEL
LIN {X 0,Y 325.321,Z 755.484,A -85,B 0,C 180,E1 13027.731,E2 13027.731} C_VEL
LIN {X 0,Y 328.325,Z 733.405,A -85,B 0,C 180,E1 13026.877,E2 13026.877} C_VEL
LIN {X 0,Y 330.385,Z 709.455,A -85,B 0,C 180,E1 13026.256,E2 13026.256} C_VEL
LIN {X 0,Y 341.286,Z 550.183,A -85,B 0,C 180,E1 13022.81,E2 13022.81} C_VEL
LIN {X 0,Y 340.927,Z 546.933,A -85,B 0,C 180,E1 13022.604,E2 13022.604} C_VEL
LIN {X 0,Y 339.151,Z 543.422,A -85,B 0,C 180,E1 13022.058,E2 13022.058} C_VEL
LIN {X 0,Y 332.496,Z 536.745,A -85,B 0,C 180,E1 13020.164,E2 13020.164} C_VEL
LIN {X 0,Y 331.881,Z 535.75,A -85,B 0,C 180,E1 13019.965,E2 13019.965} C_VEL
LIN {X 0,Y 323.332,Z 521.656,A -85,B 0,C 180,E1 13017.023,E2 13017.023} C_VEL
LIN {X 0,Y 314.496,Z 508.127,A -85,B 0,C 180,E1 13013.625,E2 13013.625} C_VEL
LIN {X 0,Y 307.45,Z 498.248,A -85,B 0,C 180,E1 13010.583,E2 13010.583} C_VEL
LIN {X 0,Y 301.596,Z 490.156,A -85,B 0,C 180,E1 13007.743,E2 13007.743} C_VEL
LIN {X 0,Y 294.407,Z 480.778,A -85,B 0,C 180,E1 13003.72,E2 13003.72} C_VEL
LIN {X 0,Y 290.509,Z 475.834,A -85,B 0,C 180,E1 13001.166,E2 13001.166} C_VEL
LIN {X 0,Y 285.893,Z 470.322,A -85,B 0,C 180,E1 12997.737,E2 12997.737} C_VEL
LIN {X 0,Y 284.258,Z 468.497,A -85,B 0,C 180,E1 12996.338,E2 12996.338} C_VEL
LIN {X 0,Y 280.652,Z 464.033,A -85,B 0,C 180,E1 12992.772,E2 12992.772} C_VEL
LIN {X 0,Y 275.238,Z 457.774,A -85,B 0,C 180,E1 12984.465,E2 12984.465} C_VEL
LIN {X 0,Y 273.672,Z 456.522,A -85,B 0,C 180,E1 12978.313,E2 12978.313} C_VEL
LIN {X 0,Y 274.17,Z 456.93,A -85,B 0,C 180,E1 12972.426,E2 12972.426} C_VEL
LIN {X 0,Y 275.612,Z 458.261,A -85,B 0,C 180,E1 12968.344,E2 12968.344} C_VEL
LIN {X 0,Y 281.094,Z 464.432,A -85,B 0,C 180,E1 12960.51,E2 12960.51} C_VEL
LIN {X 0,Y 285.02,Z 469.157,A -85,B 0,C 180,E1 12956.682,E2 12956.682} C_VEL
LIN {X 0,Y 286.349,Z 470.668,A -85,B 0,C 180,E1 12955.595,E2 12955.595} C_VEL
LIN {X 0,Y 290.082,Z 475.182,A -85,B 0,C 180,E1 12952.773,E2 12952.773} C_VEL
LIN {X 0,Y 292.288,Z 478.147,A -85,B 0,C 180,E1 12951.245,E2 12951.245} C_VEL
LIN {X 0,Y 296.118,Z 482.679,A -85,B 0,C 180,E1 12948.904,E2 12948.904} C_VEL
LIN {X 0,Y 303.219,Z 491.679,A -85,B 0,C 180,E1 12945.042,E2 12945.042} C_VEL
LIN {X 0,Y 311.511,Z 502.996,A -85,B 0,C 180,E1 12941.182,E2 12941.182} C_VEL
LIN {X 0,Y 320.323,Z 515.628,A -85,B 0,C 180,E1 12937.617,E2 12937.617} C_VEL
LIN {X 0,Y 329.377,Z 529.565,A -85,B 0,C 180,E1 12934.369,E2 12934.369} C_VEL
LIN {X 0,Y 338.056,Z 543.881,A -85,B 0,C 180,E1 12931.564,E2 12931.564} C_VEL
LIN {X 0,Y 341.658,Z 550.357,A -85,B 0,C 180,E1 12930.462,E2 12930.462} C_VEL
LIN {X 0,Y 328.481,Z 750.562,A -85,B 0,C 180,E1 12926.213,E2 12926.213} C_VEL
LIN {X 0,Y 325.601,Z 772.668,A -85,B 0,C 180,E1 12925.529,E2 12925.529} C_VEL
LIN {X 0,Y 321.663,Z 794.198,A -85,B 0,C 180,E1 12924.609,E2 12924.609} C_VEL
LIN {X 0,Y 316.918,Z 815.102,A -85,B 0,C 180,E1 12923.415,E2 12923.415} C_VEL
LIN {X 0,Y 311.591,Z 834.839,A -85,B 0,C 180,E1 12921.968,E2 12921.968} C_VEL
LIN {X 0,Y 305.703,Z 853.636,A -85,B 0,C 180,E1 12920.233,E2 12920.233} C_VEL
LIN {X 0,Y 298.821,Z 873.269,A -85,B 0,C 180,E1 12917.995,E2 12917.995} C_VEL
LIN {X 0,Y 292.159,Z 890.77,A -85,B 0,C 180,E1 12915.529,E2 12915.529} C_VEL
LIN {X 0,Y 285.267,Z 907.676,A -85,B 0,C 180,E1 12912.605,E2 12912.605} C_VEL
LIN {X 0,Y 278.807,Z 922.718,A -85,B 0,C 180,E1 12909.406,E2 12909.406} C_VEL
LIN {X 0,Y 272.928,Z 936.359,A -85,B 0,C 180,E1 12905.889,E2 12905.889} C_VEL
LIN {X 0,Y 267.716,Z 948.716,A -85,B 0,C 180,E1 12902.029,E2 12902.029} C_VEL
LIN {X 0,Y 263.331,Z 959.729,A -85,B 0,C 180,E1 12897.788,E2 12897.788} C_VEL
LIN {X 0,Y 260.047,Z 969.04,A -85,B 0,C 180,E1 12893.334,E2 12893.334} C_VEL
LIN {X 0,Y 257.815,Z 976.984,A -85,B 0,C 180,E1 12888.547,E2 12888.547} C_VEL
LIN {X 0,Y 256.715,Z 982.819,A -85,B 0,C 180,E1 12883.978,E2 12883.978} C_VEL
LIN {X 0,Y 256.373,Z 986.731,A -85,B 0,C 180,E1 12879.659,E2 12879.659} C_VEL
LIN {X 0,Y 256.436,Z 989.208,A -85,B 0,C 180,E1 12875.598,E2 12875.598} C_VEL
LIN {X 0,Y 256.562,Z 990.346,A -85,B 0,C 180,E1 12871.345,E2 12871.345} C_VEL
LIN {X 0,Y 256.537,Z 990.231,A -85,B 0,C 180,E1 12867.771,E2 12867.771} C_VEL
LIN {X 0,Y 256.407,Z 988.833,A -85,B 0,C 180,E1 12863.512,E2 12863.512} C_VEL
LIN {X 0,Y 256.411,Z 985.953,A -85,B 0,C 180,E1 12859.217,E2 12859.217} C_VEL
LIN {X 0,Y 256.973,Z 981.197,A -85,B 0,C 180,E1 12854.432,E2 12854.432} C_VEL
LIN {X 0,Y 258.408,Z 975.039,A -85,B 0,C 180,E1 12849.862,E2 12849.862} C_VEL
LIN {X 0,Y 260.975,Z 966.981,A -85,B 0,C 180,E1 12845.23,E2 12845.23} C_VEL
LIN {X 0,Y 264.876,Z 956.972,A -85,B 0,C 180,E1 12840.618,E2 12840.618} C_VEL
LIN {X 0,Y 269.71,Z 945.955,A -85,B 0,C 180,E1 12836.477,E2 12836.477} C_VEL
LIN {X 0,Y 275.439,Z 933.404,A -85,B 0,C 180,E1 12832.653,E2 12832.653} C_VEL
LIN {X 0,Y 282.344,Z 918.675,A -85,B 0,C 180,E1 12828.963,E2 12828.963} C_VEL
LIN {X 0,Y 289.529,Z 903.086,A -85,B 0,C 180,E1 12825.774,E2 12825.774} C_VEL
LIN {X 0,Y 296.946,Z 886.382,A -85,B 0,C 180,E1 12822.977,E2 12822.977} C_VEL
LIN {X 0,Y 304.164,Z 868.836,A -85,B 0,C 180,E1 12820.601,E2 12820.601} C_VEL
LIN {X 0,Y 311.513,Z 849.364,A -85,B 0,C 180,E1 12818.458,E2 12818.458} C_VEL
LIN {X 0,Y 318.117,Z 829.822,A -85,B 0,C 180,E1 12816.737,E2 12816.737} C_VEL
LIN {X 0,Y 324.081,Z 809.432,A -85,B 0,C 180,E1 12815.319,E2 12815.319} C_VEL
LIN {X 0,Y 329.176,Z 788.461,A -85,B 0,C 180,E1 12814.205,E2 12814.205} C_VEL
LIN {X 0,Y 333.4,Z 766.675,A -85,B 0,C 180,E1 12813.352,E2 12813.352} C_VEL
LIN {X 0,Y 336.366,Z 744.537,A -85,B 0,C 180,E1 12812.71,E2 12812.71} C_VEL
LIN {X 0,Y 351.401,Z 552.89,A -85,B 0,C 180,E1 12808.583,E2 12808.583} C_VEL
LIN {X 0,Y 346.439,Z 542.807,A -85,B 0,C 180,E1 12806.162,E2 12806.162} C_VEL
LIN {X 0,Y 341.744,Z 534.128,A -85,B 0,C 180,E1 12803.447,E2 12803.447} C_VEL
LIN {X 0,Y 337.788,Z 527.154,A -85,B 0,C 180,E1 12800.533,E2 12800.533} C_VEL
LIN {X 0,Y 334.951,Z 522.581,A -85,B 0,C 180,E1 12797.726,E2 12797.726} C_VEL
LIN {X 0,Y 332.523,Z 518.426,A -85,B 0,C 180,E1 12793.387,E2 12793.387} C_VEL
LIN {X 0,Y 332.24,Z 518.178,A -85,B 0,C 180,E1 12789.527,E2 12789.527} C_VEL
LIN {X 0,Y 332.646,Z 518.942,A -85,B 0,C 180,E1 12787.947,E2 12787.947} C_VEL
LIN {X 0,Y 335.061,Z 523.221,A -85,B 0,C 180,E1 12783.849,E2 12783.849} C_VEL
LIN {X 0,Y 338.029,Z 528.427,A -85,B 0,C 180,E1 12780.94,E2 12780.94} C_VEL
LIN {X 0,Y 341.644,Z 534.97,A -85,B 0,C 180,E1 12778.281,E2 12778.281} C_VEL
LIN {X 0,Y 346.029,Z 543.171,A -85,B 0,C 180,E1 12775.691,E2 12775.691} C_VEL
LIN {X 0,Y 350.237,Z 552.014,A -85,B 0,C 180,E1 12773.555,E2 12773.555} C_VEL
LIN {X 0,Y 334.436,Z 731.256,A -85,B 0,C 180,E1 12769.567,E2 12769.567} C_VEL
LIN {X 0,Y 331.456,Z 751.947,A -85,B 0,C 180,E1 12768.847,E2 12768.847} C_VEL
LIN {X 0,Y 327.637,Z 771.58,A -85,B 0,C 180,E1 12767.912,E2 12767.912} C_VEL
LIN {X 0,Y 322.657,Z 792.012,A -85,B 0,C 180,E1 12766.64,E2 12766.64} C_VEL
LIN {X 0,Y 317.088,Z 810.98,A -85,B 0,C 180,E1 12765.135,E2 12765.135} C_VEL
LIN {X 0,Y 310.607,Z 829.842,A -85,B 0,C 180,E1 12763.249,E2 12763.249} C_VEL
LIN {X 0,Y 303.82,Z 847.134,A -85,B 0,C 180,E1 12761.094,E2 12761.094} C_VEL
LIN {X 0,Y 296.985,Z 862.897,A -85,B 0,C 180,E1 12758.678,E2 12758.678} C_VEL
LIN {X 0,Y 289.575,Z 878.613,A -85,B 0,C 180,E1 12755.706,E2 12755.706} C_VEL
LIN {X 0,Y 282.802,Z 892.151,A -85,B 0,C 180,E1 12752.538,E2 12752.538} C_VEL
LIN {X 0,Y 276.629,Z 904.009,A -85,B 0,C 180,E1 12749.119,E2 12749.119} C_VEL
LIN {X 0,Y 270.673,Z 915.184,A -85,B 0,C 180,E1 12745.08,E2 12745.08} C_VEL
LIN {X 0,Y 265.768,Z 924.436,A -85,B 0,C 180,E1 12740.796,E2 12740.796} C_VEL
LIN {X 0,Y 262.096,Z 931.687,A -85,B 0,C 180,E1 12736.445,E2 12736.445} C_VEL
LIN {X 0,Y 259.428,Z 937.441,A -85,B 0,C 180,E1 12731.809,E2 12731.809} C_VEL
LIN {X 0,Y 257.853,Z 941.38,A -85,B 0,C 180,E1 12727.215,E2 12727.215} C_VEL
LIN {X 0,Y 257.064,Z 943.703,A -85,B 0,C 180,E1 12722.721,E2 12722.721} C_VEL
LIN {X 0,Y 256.773,Z 944.44,A -85,B 0,C 180,E1 12718.352,E2 12718.352} C_VEL
LIN {X 0,Y 256.797,Z 943.777,A -85,B 0,C 180,E1 12713.794,E2 12713.794} C_VEL
LIN {X 0,Y 257.168,Z 941.821,A -85,B 0,C 180,E1 12709.528,E2 12709.528} C_VEL
LIN {X 0,Y 258.069,Z 938.163,A -85,B 0,C 180,E1 12705.04,E2 12705.04} C_VEL
LIN {X 0,Y 259.746,Z 932.992,A -85,B 0,C 180,E1 12700.643,E2 12700.643} C_VEL
LIN {X 0,Y 262.496,Z 925.838,A -85,B 0,C 180,E1 12696.118,E2 12696.118} C_VEL
LIN {X 0,Y 266.13,Z 917.284,A -85,B 0,C 180,E1 12691.933,E2 12691.933} C_VEL
LIN {X 0,Y 270.785,Z 906.824,A -85,B 0,C 180,E1 12687.879,E2 12687.879} C_VEL
LIN {X 0,Y 276.142,Z 894.847,A -85,B 0,C 180,E1 12684.177,E2 12684.177} C_VEL
LIN {X 0,Y 281.635,Z 882.246,A -85,B 0,C 180,E1 12681.009,E2 12681.009} C_VEL
LIN {X 0,Y 287.834,Z 867.489,A -85,B 0,C 180,E1 12677.966,E2 12677.966} C_VEL
LIN {X 0,Y 293.999,Z 851.793,A -85,B 0,C 180,E1 12675.319,E2 12675.319} C_VEL
LIN {X 0,Y 300.096,Z 834.868,A -85,B 0,C 180,E1 12672.987,E2 12672.987} C_VEL
LIN {X 0,Y 306.053,Z 816.367,A -85,B 0,C 180,E1 12670.928,E2 12670.928} C_VEL
LIN {X 0,Y 311.395,Z 797.128,A -85,B 0,C 180,E1 12669.215,E2 12669.215} C_VEL
LIN {X 0,Y 315.855,Z 778.092,A -85,B 0,C 180,E1 12667.867,E2 12667.867} C_VEL
LIN {X 0,Y 319.968,Z 756.438,A -85,B 0,C 180,E1 12666.688,E2 12666.688} C_VEL
LIN {X 0,Y 323.05,Z 734.757,A -85,B 0,C 180,E1 12665.834,E2 12665.834} C_VEL
LIN {X 0,Y 325.132,Z 712.149,A -85,B 0,C 180,E1 12665.231,E2 12665.231} C_VEL
LIN {X 0,Y 336.965,Z 544.809,A -85,B 0,C 180,E1 12661.594,E2 12661.594} C_VEL
LIN {X 0,Y 331.881,Z 535.75,A -85,B 0,C 180,E1 12659.965,E2 12659.965} C_VEL
LIN {X 0,Y 329.192,Z 532.191,A -85,B 0,C 180,E1 12659.111,E2 12659.111} C_VEL
LIN {X 0,Y 323.963,Z 528.401,A -85,B 0,C 180,E1 12657.509,E2 12657.509} C_VEL
LIN {X 0,Y 318.341,Z 524.48,A -85,B 0,C 180,E1 12655.662,E2 12655.662} C_VEL
LIN {X 0,Y 316.191,Z 521.811,A -85,B 0,C 180,E1 12654.861,E2 12654.861} C_VEL
LIN {X 0,Y 309.184,Z 511.27,A -85,B 0,C 180,E1 12651.948,E2 12651.948} C_VEL
LIN {X 0,Y 302.696,Z 502.024,A -85,B 0,C 180,E1 12648.935,E2 12648.935} C_VEL
LIN {X 0,Y 296.306,Z 493.215,A -85,B 0,C 180,E1 12645.537,E2 12645.537} C_VEL
LIN {X 0,Y 291.782,Z 487.495,A -85,B 0,C 180,E1 12642.83,E2 12642.83} C_VEL
LIN {X 0,Y 287.868,Z 482.357,A -85,B 0,C 180,E1 12640.127,E2 12640.127} C_VEL
LIN {X 0,Y 284.18,Z 477.737,A -85,B 0,C 180,E1 12637.241,E2 12637.241} C_VEL
LIN {X 0,Y 279.189,Z 471.636,A -85,B 0,C 180,E1 12632.36,E2 12632.36} C_VEL
LIN {X 0,Y 274.041,Z 465.6,A -85,B 0,C 180,E1 12624.12,E2 12624.12} C_VEL
LIN {X 0,Y 272.609,Z 464.448,A -85,B 0,C 180,E1 12618.166,E2 12618.166} C_VEL
LIN {X 0,Y 273.097,Z 464.855,A -85,B 0,C 180,E1 12612.475,E2 12612.475} C_VEL
LIN {X 0,Y 274.433,Z 466.085,A -85,B 0,C 180,E1 12608.591,E2 12608.591} C_VEL
LIN {X 0,Y 279.791,Z 472.321,A -85,B 0,C 180,E1 12600.717,E2 12600.717} C_VEL
LIN {X 0,Y 283.698,Z 476.999,A -85,B 0,C 180,E1 12596.869,E2 12596.869} C_VEL
LIN {X 0,Y 285.224,Z 479.04,A -85,B 0,C 180,E1 12595.577,E2 12595.577} C_VEL
LIN {X 0,Y 289.561,Z 484.24,A -85,B 0,C 180,E1 12592.332,E2 12592.332} C_VEL
LIN {X 0,Y 294.449,Z 490.477,A -85,B 0,C 180,E1 12589.187,E2 12589.187} C_VEL
LIN {X 0,Y 301.029,Z 498.978,A -85,B 0,C 180,E1 12585.527,E2 12585.527} C_VEL
LIN {X 0,Y 309.038,Z 510.063,A -85,B 0,C 180,E1 12581.71,E2 12581.71} C_VEL
LIN {X 0,Y 317.408,Z 522.257,A -85,B 0,C 180,E1 12578.228,E2 12578.228} C_VEL
LIN {X 0,Y 326.319,Z 536.213,A -85,B 0,C 180,E1 12574.938,E2 12574.938} C_VEL
LIN {X 0,Y 335.466,Z 551.591,A -85,B 0,C 180,E1 12571.906,E2 12571.906} C_VEL
LIN {X 0,Y 336.758,Z 554.258,A -85,B 0,C 180,E1 12571.485,E2 12571.485} C_VEL
LIN {X 0,Y 323.399,Z 750.21,A -85,B 0,C 180,E1 12567.306,E2 12567.306} C_VEL
LIN {X 0,Y 320.438,Z 772.36,A -85,B 0,C 180,E1 12566.619,E2 12566.619} C_VEL
LIN {X 0,Y 316.459,Z 793.56,A -85,B 0,C 180,E1 12565.716,E2 12565.716} C_VEL
LIN {X 0,Y 311.534,Z 814.69,A -85,B 0,C 180,E1 12564.511,E2 12564.511} C_VEL
LIN {X 0,Y 305.974,Z 834.669,A -85,B 0,C 180,E1 12563.04,E2 12563.04} C_VEL
LIN {X 0,Y 299.868,Z 853.49,A -85,B 0,C 180,E1 12561.286,E2 12561.286} C_VEL
LIN {X 0,Y 292.963,Z 872.52,A -85,B 0,C 180,E1 12559.099,E2 12559.099} C_VEL
LIN {X 0,Y 286.102,Z 889.918,A -85,B 0,C 180,E1 12556.632,E2 12556.632} C_VEL
LIN {X 0,Y 279.089,Z 906.479,A -85,B 0,C 180,E1 12553.748,E2 12553.748} C_VEL
LIN {X 0,Y 272.375,Z 921.536,A -85,B 0,C 180,E1 12550.527,E2 12550.527} C_VEL
LIN {X 0,Y 265.833,Z 936.002,A -85,B 0,C 180,E1 12546.734,E2 12546.734} C_VEL
LIN {X 0,Y 260.309,Z 948.436,A -85,B 0,C 180,E1 12542.735,E2 12542.735} C_VEL
LIN {X 0,Y 255.598,Z 959.722,A -85,B 0,C 180,E1 12538.255,E2 12538.255} C_VEL
LIN {X 0,Y 252.144,Z 969.008,A -85,B 0,C 180,E1 12533.614,E2 12533.614} C_VEL
LIN {X 0,Y 249.838,Z 976.79,A -85,B 0,C 180,E1 12528.677,E2 12528.677} C_VEL
LIN {X 0,Y 248.717,Z 982.495,A -85,B 0,C 180,E1 12523.962,E2 12523.962} C_VEL
LIN {X 0,Y 248.39,Z 986.298,A -85,B 0,C 180,E1 12519.504,E2 12519.504} C_VEL
LIN {X 0,Y 248.474,Z 988.748,A -85,B 0,C 180,E1 12515.084,E2 12515.084} C_VEL
LIN {X 0,Y 248.597,Z 989.643,A -85,B 0,C 180,E1 12511.157,E2 12511.157} C_VEL
LIN {X 0,Y 248.551,Z 989.449,A -85,B 0,C 180,E1 12507.238,E2 12507.238} C_VEL
LIN {X 0,Y 248.395,Z 987.869,A -85,B 0,C 180,E1 12502.837,E2 12502.837} C_VEL
LIN {X 0,Y 248.45,Z 985.065,A -85,B 0,C 180,E1 12498.632,E2 12498.632} C_VEL
LIN {X 0,Y 249.172,Z 980.052,A -85,B 0,C 180,E1 12493.542,E2 12493.542} C_VEL
LIN {X 0,Y 250.876,Z 973.685,A -85,B 0,C 180,E1 12488.741,E2 12488.741} C_VEL
LIN {X 0,Y 253.895,Z 965.173,A -85,B 0,C 180,E1 12483.834,E2 12483.834} C_VEL
LIN {X 0,Y 258.108,Z 955.255,A -85,B 0,C 180,E1 12479.253,E2 12479.253} C_VEL
LIN {X 0,Y 263.394,Z 944.035,A -85,B 0,C 180,E1 12475.033,E2 12475.033} C_VEL
LIN {X 0,Y 269.927,Z 930.757,A -85,B 0,C 180,E1 12470.978,E2 12470.978} C_VEL
LIN {X 0,Y 276.984,Z 916.38,A -85,B 0,C 180,E1 12467.425,E2 12467.425} C_VEL
LIN {X 0,Y 284.885,Z 900.038,A -85,B 0,C 180,E1 12464.135,E2 12464.135} C_VEL
LIN {X 0,Y 292.598,Z 883.219,A -85,B 0,C 180,E1 12461.383,E2 12461.383} C_VEL
LIN {X 0,Y 300.321,Z 865.193,A -85,B 0,C 180,E1 12458.993,E2 12458.993} C_VEL
LIN {X 0,Y 307.431,Z 846.719,A -85,B 0,C 180,E1 12457.028,E2 12457.028} C_VEL
LIN {X 0,Y 314.307,Z 826.785,A -85,B 0,C 180,E1 12455.326,E2 12455.326} C_VEL
LIN {X 0,Y 320.324,Z 806.608,A -85,B 0,C 180,E1 12453.967,E2 12453.967} C_VEL
LIN {X 0,Y 325.408,Z 786.078,A -85,B 0,C 180,E1 12452.912,E2 12452.912} C_VEL
LIN {X 0,Y 329.591,Z 764.542,A -85,B 0,C 180,E1 12452.097,E2 12452.097} C_VEL
LIN {X 0,Y 332.633,Z 741.449,A -85,B 0,C 180,E1 12451.448,E2 12451.448} C_VEL
LIN {X 0,Y 347.705,Z 557.155,A -85,B 0,C 180,E1 12447.469,E2 12447.469} C_VEL
LIN {X 0,Y 343.199,Z 547.888,A -85,B 0,C 180,E1 12445.08,E2 12445.08} C_VEL
LIN {X 0,Y 339.079,Z 540.076,A -85,B 0,C 180,E1 12442.449,E2 12442.449} C_VEL
LIN {X 0,Y 335.943,Z 534.341,A -85,B 0,C 180,E1 12439.924,E2 12439.924} C_VEL
LIN {X 0,Y 333.603,Z 530.312,A -85,B 0,C 180,E1 12437.44,E2 12437.44} C_VEL
LIN {X 0,Y 331.411,Z 526.32,A -85,B 0,C 180,E1 12433.255,E2 12433.255} C_VEL
LIN {X 0,Y 331.187,Z 526.15,A -85,B 0,C 180,E1 12429.382,E2 12429.382} C_VEL
LIN {X 0,Y 331.588,Z 527.136,A -85,B 0,C 180,E1 12427.798,E2 12427.798} C_VEL
LIN {X 0,Y 333.714,Z 530.968,A -85,B 0,C 180,E1 12424.123,E2 12424.123} C_VEL
LIN {X 0,Y 336.455,Z 536.034,A -85,B 0,C 180,E1 12421.277,E2 12421.277} C_VEL
LIN {X 0,Y 339.924,Z 542.638,A -85,B 0,C 180,E1 12418.609,E2 12418.609} C_VEL
LIN {X 0,Y 343.937,Z 550.53,A -85,B 0,C 180,E1 12416.124,E2 12416.124} C_VEL
LIN {X 0,Y 346.607,Z 556.451,A -85,B 0,C 180,E1 12414.669,E2 12414.669} C_VEL
LIN {X 0,Y 330.547,Z 731.643,A -85,B 0,C 180,E1 12410.771,E2 12410.771} C_VEL
LIN {X 0,Y 327.409,Z 752.675,A -85,B 0,C 180,E1 12410.041,E2 12410.041} C_VEL
LIN {X 0,Y 323.331,Z 772.875,A -85,B 0,C 180,E1 12409.077,E2 12409.077} C_VEL
LIN {X 0,Y 318.116,Z 793.316,A -85,B 0,C 180,E1 12407.794,E2 12407.794} C_VEL
LIN {X 0,Y 312.365,Z 812.03,A -85,B 0,C 180,E1 12406.298,E2 12406.298} C_VEL
LIN {X 0,Y 305.77,Z 830.513,A -85,B 0,C 180,E1 12404.446,E2 12404.446} C_VEL
LIN {X 0,Y 298.625,Z 847.968,A -85,B 0,C 180,E1 12402.26,E2 12402.26} C_VEL
LIN {X 0,Y 291.346,Z 863.998,A -85,B 0,C 180,E1 12399.775,E2 12399.775} C_VEL
LIN {X 0,Y 283.789,Z 879.308,A -85,B 0,C 180,E1 12396.847,E2 12396.847} C_VEL
LIN {X 0,Y 276.583,Z 892.973,A -85,B 0,C 180,E1 12393.598,E2 12393.598} C_VEL
LIN {X 0,Y 269.969,Z 905.013,A -85,B 0,C 180,E1 12390.059,E2 12390.059} C_VEL
LIN {X 0,Y 263.865,Z 915.794,A -85,B 0,C 180,E1 12386.073,E2 12386.073} C_VEL
LIN {X 0,Y 258.748,Z 924.837,A -85,B 0,C 180,E1 12381.809,E2 12381.809} C_VEL
LIN {X 0,Y 254.881,Z 931.925,A -85,B 0,C 180,E1 12377.509,E2 12377.509} C_VEL
LIN {X 0,Y 251.901,Z 937.822,A -85,B 0,C 180,E1 12372.737,E2 12372.737} C_VEL
LIN {X 0,Y 250.1,Z 941.907,A -85,B 0,C 180,E1 12367.993,E2 12367.993} C_VEL
LIN {X 0,Y 249.169,Z 944.289,A -85,B 0,C 180,E1 12363.343,E2 12363.343} C_VEL
LIN {X 0,Y 248.822,Z 945.148,A -85,B 0,C 180,E1 12358.823,E2 12358.823} C_VEL
LIN {X 0,Y 248.813,Z 944.718,A -85,B 0,C 180,E1 12354.444,E2 12354.444} C_VEL
LIN {X 0,Y 249.14,Z 942.843,A -85,B 0,C 180,E1 12349.94,E2 12349.94} C_VEL
LIN {X 0,Y 250.029,Z 939.385,A -85,B 0,C 180,E1 12345.298,E2 12345.298} C_VEL
LIN {X 0,Y 251.821,Z 934.124,A -85,B 0,C 180,E1 12340.518,E2 12340.518} C_VEL
LIN {X 0,Y 254.502,Z 927.514,A -85,B 0,C 180,E1 12336.084,E2 12336.084} C_VEL
LIN {X 0,Y 258.21,Z 919.17,A -85,B 0,C 180,E1 12331.77,E2 12331.77} C_VEL
LIN {X 0,Y 262.968,Z 908.891,A -85,B 0,C 180,E1 12327.598,E2 12327.598} C_VEL
LIN {X 0,Y 268.46,Z 897.18,A -85,B 0,C 180,E1 12323.795,E2 12323.795} C_VEL
LIN {X 0,Y 274.482,Z 884.069,A -85,B 0,C 180,E1 12320.35,E2 12320.35} C_VEL
LIN {X 0,Y 280.906,Z 869.486,A -85,B 0,C 180,E1 12317.236,E2 12317.236} C_VEL
LIN {X 0,Y 287.255,Z 854.107,A -85,B 0,C 180,E1 12314.553,E2 12314.553} C_VEL
LIN {X 0,Y 293.87,Z 836.489,A -85,B 0,C 180,E1 12312.063,E2 12312.063} C_VEL
LIN {X 0,Y 300.167,Z 817.622,A -85,B 0,C 180,E1 12309.931,E2 12309.931} C_VEL
LIN {X 0,Y 305.413,Z 799.499,A -85,B 0,C 180,E1 12308.285,E2 12308.285} C_VEL
LIN {X 0,Y 310.284,Z 779.692,A -85,B 0,C 180,E1 12306.847,E2 12306.847} C_VEL
LIN {X 0,Y 314.418,Z 758.982,A -85,B 0,C 180,E1 12305.689,E2 12305.689} C_VEL
LIN {X 0,Y 317.645,Z 737.824,A -85,B 0,C 180,E1 12304.818,E2 12304.818} C_VEL
LIN {X 0,Y 319.888,Z 715.567,A -85,B 0,C 180,E1 12304.196,E2 12304.196} C_VEL
LIN {X 0,Y 332.056,Z 548.462,A -85,B 0,C 180,E1 12300.528,E2 12300.528} C_VEL
LIN {X 0,Y 323.589,Z 533.674,A -85,B 0,C 180,E1 12297.637,E2 12297.637} C_VEL
LIN {X 0,Y 316.191,Z 521.811,A -85,B 0,C 180,E1 12294.861,E2 12294.861} C_VEL
LIN {X 0,Y 313.643,Z 518.871,A -85,B 0,C 180,E1 12293.879,E2 12293.879} C_VEL
LIN {X 0,Y 308.825,Z 516.212,A -85,B 0,C 180,E1 12292.085,E2 12292.085} C_VEL
LIN {X 0,Y 303.767,Z 513.458,A -85,B 0,C 180,E1 12290.032,E2 12290.032} C_VEL
LIN {X 0,Y 301.834,Z 511.223,A -85,B 0,C 180,E1 12289.133,E2 12289.133} C_VEL
LIN {X 0,Y 295.842,Z 502.821,A -85,B 0,C 180,E1 12285.975,E2 12285.975} C_VEL
LIN {X 0,Y 290.094,Z 495.135,A -85,B 0,C 180,E1 12282.497,E2 12282.497} C_VEL
LIN {X 0,Y 286.039,Z 489.811,A -85,B 0,C 180,E1 12279.639,E2 12279.639} C_VEL
LIN {X 0,Y 282.375,Z 484.94,A -85,B 0,C 180,E1 12276.63,E2 12276.63} C_VEL
LIN {X 0,Y 278.031,Z 479.773,A -85,B 0,C 180,E1 12272.311,E2 12272.311} C_VEL
LIN {X 0,Y 273.01,Z 473.575,A -85,B 0,C 180,E1 12264.217,E2 12264.217} C_VEL
LIN {X 0,Y 271.544,Z 472.378,A -85,B 0,C 180,E1 12258.189,E2 12258.189} C_VEL
LIN {X 0,Y 272.023,Z 472.78,A -85,B 0,C 180,E1 12252.525,E2 12252.525} C_VEL
LIN {X 0,Y 273.348,Z 474.066,A -85,B 0,C 180,E1 12248.626,E2 12248.626} C_VEL
LIN {X 0,Y 278.402,Z 480.064,A -85,B 0,C 180,E1 12241.03,E2 12241.03} C_VEL
LIN {X 0,Y 282.335,Z 484.805,A -85,B 0,C 180,E1 12237.094,E2 12237.094} C_VEL
LIN {X 0,Y 287.083,Z 490.677,A -85,B 0,C 180,E1 12233.3,E2 12233.3} C_VEL
LIN {X 0,Y 292.711,Z 498.172,A -85,B 0,C 180,E1 12229.52,E2 12229.52} C_VEL
LIN {X 0,Y 298.87,Z 506.286,A -85,B 0,C 180,E1 12226.013,E2 12226.013} C_VEL
LIN {X 0,Y 306.494,Z 517.015,A -85,B 0,C 180,E1 12222.276,E2 12222.276} C_VEL
LIN {X 0,Y 314.598,Z 529.048,A -85,B 0,C 180,E1 12218.807,E2 12218.807} C_VEL
LIN {X 0,Y 323.273,Z 542.855,A -85,B 0,C 180,E1 12215.516,E2 12215.516} C_VEL
LIN {X 0,Y 331.97,Z 557.819,A -85,B 0,C 180,E1 12212.543,E2 12212.543} C_VEL
LIN {X 0,Y 318.411,Z 749.793,A -85,B 0,C 180,E1 12208.43,E2 12208.43} C_VEL
LIN {X 0,Y 315.383,Z 771.888,A -85,B 0,C 180,E1 12207.744,E2 12207.744} C_VEL
LIN {X 0,Y 311.3,Z 793.062,A -85,B 0,C 180,E1 12206.845,E2 12206.845} C_VEL
LIN {X 0,Y 306.348,Z 813.779,A -85,B 0,C 180,E1 12205.668,E2 12205.668} C_VEL
LIN {X 0,Y 300.724,Z 833.482,A -85,B 0,C 180,E1 12204.224,E2 12204.224} C_VEL
LIN {X 0,Y 294.449,Z 852.378,A -85,B 0,C 180,E1 12202.475,E2 12202.475} C_VEL
LIN {X 0,Y 287.313,Z 871.534,A -85,B 0,C 180,E1 12200.276,E2 12200.276} C_VEL
LIN {X 0,Y 280.414,Z 888.481,A -85,B 0,C 180,E1 12197.877,E2 12197.877} C_VEL
LIN {X 0,Y 272.952,Z 905.398,A -85,B 0,C 180,E1 12194.913,E2 12194.913} C_VEL
LIN {X 0,Y 266.049,Z 920.295,A -85,B 0,C 180,E1 12191.702,E2 12191.702} C_VEL
LIN {X 0,Y 259.143,Z 934.888,A -85,B 0,C 180,E1 12187.846,E2 12187.846} C_VEL
LIN {X 0,Y 253.364,Z 947.282,A -85,B 0,C 180,E1 12183.814,E2 12183.814} C_VEL
LIN {X 0,Y 248.491,Z 958.199,A -85,B 0,C 180,E1 12179.404,E2 12179.404} C_VEL
LIN {X 0,Y 244.701,Z 967.663,A -85,B 0,C 180,E1 12174.636,E2 12174.636} C_VEL
LIN {X 0,Y 242.113,Z 975.616,A -85,B 0,C 180,E1 12169.547,E2 12169.547} C_VEL
LIN {X 0,Y 240.829,Z 981.456,A -85,B 0,C 180,E1 12164.675,E2 12164.675} C_VEL
LIN {X 0,Y 240.419,Z 985.354,A -85,B 0,C 180,E1 12160.064,E2 12160.064} C_VEL
LIN {X 0,Y 240.492,Z 987.931,A -85,B 0,C 180,E1 12155.492,E2 12155.492} C_VEL
LIN {X 0,Y 240.628,Z 988.919,A -85,B 0,C 180,E1 12151.195,E2 12151.195} C_VEL
LIN {X 0,Y 240.585,Z 988.767,A -85,B 0,C 180,E1 12147.385,E2 12147.385} C_VEL
LIN {X 0,Y 240.414,Z 987.3,A -85,B 0,C 180,E1 12142.838,E2 12142.838} C_VEL
LIN {X 0,Y 240.482,Z 984.371,A -85,B 0,C 180,E1 12138.25,E2 12138.25} C_VEL
LIN {X 0,Y 241.265,Z 979.548,A -85,B 0,C 180,E1 12133.142,E2 12133.142} C_VEL
LIN {X 0,Y 243.17,Z 973.013,A -85,B 0,C 180,E1 12128.033,E2 12128.033} C_VEL
LIN {X 0,Y 246.443,Z 964.527,A -85,B 0,C 180,E1 12122.98,E2 12122.98} C_VEL
LIN {X 0,Y 251.235,Z 954.09,A -85,B 0,C 180,E1 12118.048,E2 12118.048} C_VEL
LIN {X 0,Y 257.257,Z 942.139,A -85,B 0,C 180,E1 12113.519,E2 12113.519} C_VEL
LIN {X 0,Y 264.297,Z 928.701,A -85,B 0,C 180,E1 12109.414,E2 12109.414} C_VEL
LIN {X 0,Y 272.114,Z 913.683,A -85,B 0,C 180,E1 12105.73,E2 12105.73} C_VEL
LIN {X 0,Y 279.952,Z 898.098,A -85,B 0,C 180,E1 12102.639,E2 12102.639} C_VEL
LIN {X 0,Y 288.289,Z 880.573,A -85,B 0,C 180,E1 12099.815,E2 12099.815} C_VEL
LIN {X 0,Y 296.162,Z 862.798,A -85,B 0,C 180,E1 12097.507,E2 12097.507} C_VEL
LIN {X 0,Y 303.573,Z 844.206,A -85,B 0,C 180,E1 12095.568,E2 12095.568} C_VEL
LIN {X 0,Y 310.377,Z 824.854,A -85,B 0,C 180,E1 12093.96,E2 12093.96} C_VEL
LIN {X 0,Y 316.788,Z 803.716,A -85,B 0,C 180,E1 12092.582,E2 12092.582} C_VEL
LIN {X 0,Y 321.838,Z 783.838,A -85,B 0,C 180,E1 12091.59,E2 12091.59} C_VEL
LIN {X 0,Y 326.054,Z 762.182,A -85,B 0,C 180,E1 12090.799,E2 12090.799} C_VEL
LIN {X 0,Y 328.958,Z 739.96,A -85,B 0,C 180,E1 12090.191,E2 12090.191} C_VEL
LIN {X 0,Y 344.197,Z 561.655,A -85,B 0,C 180,E1 12086.341,E2 12086.341} C_VEL
LIN {X 0,Y 340.676,Z 554.136,A -85,B 0,C 180,E1 12084.306,E2 12084.306} C_VEL
LIN {X 0,Y 337.084,Z 547.016,A -85,B 0,C 180,E1 12081.845,E2 12081.845} C_VEL
LIN {X 0,Y 334.324,Z 541.783,A -85,B 0,C 180,E1 12079.478,E2 12079.478} C_VEL
LIN {X 0,Y 332.278,Z 538.044,A -85,B 0,C 180,E1 12077.151,E2 12077.151} C_VEL
LIN {X 0,Y 330.297,Z 534.213,A -85,B 0,C 180,E1 12073.122,E2 12073.122} C_VEL
LIN {X 0,Y 330.098,Z 534.075,A -85,B 0,C 180,E1 12069.413,E2 12069.413} C_VEL
LIN {X 0,Y 330.433,Z 534.968,A -85,B 0,C 180,E1 12068.001,E2 12068.001} C_VEL
LIN {X 0,Y 332.374,Z 538.712,A -85,B 0,C 180,E1 12064.399,E2 12064.399} C_VEL
LIN {X 0,Y 334.885,Z 543.621,A -85,B 0,C 180,E1 12061.625,E2 12061.625} C_VEL
LIN {X 0,Y 338.097,Z 550.054,A -85,B 0,C 180,E1 12059.025,E2 12059.025} C_VEL
LIN {X 0,Y 341.951,Z 558.069,A -85,B 0,C 180,E1 12056.521,E2 12056.521} C_VEL
LIN {X 0,Y 343.13,Z 561.009,A -85,B 0,C 180,E1 12055.805,E2 12055.805} C_VEL
LIN {X 0,Y 326.84,Z 732.347,A -85,B 0,C 180,E1 12052.001,E2 12052.001} C_VEL
LIN {X 0,Y 323.63,Z 753.137,A -85,B 0,C 180,E1 12051.283,E2 12051.283} C_VEL
LIN {X 0,Y 319.457,Z 773.1,A -85,B 0,C 180,E1 12050.337,E2 12050.337} C_VEL
LIN {X 0,Y 314.117,Z 793.353,A -85,B 0,C 180,E1 12049.076,E2 12049.076} C_VEL
LIN {X 0,Y 308.139,Z 812.256,A -85,B 0,C 180,E1 12047.579,E2 12047.579} C_VEL
LIN {X 0,Y 301.234,Z 830.87,A -85,B 0,C 180,E1 12045.721,E2 12045.721} C_VEL
LIN {X 0,Y 293.921,Z 848.03,A -85,B 0,C 180,E1 12043.577,E2 12043.577} C_VEL
LIN {X 0,Y 286.37,Z 864.078,A -85,B 0,C 180,E1 12041.101,E2 12041.101} C_VEL
LIN {X 0,Y 278.398,Z 879.525,A -85,B 0,C 180,E1 12038.142,E2 12038.142} C_VEL
LIN {X 0,Y 270.838,Z 893.229,A -85,B 0,C 180,E1 12034.877,E2 12034.877} C_VEL
LIN {X 0,Y 264.086,Z 904.883,A -85,B 0,C 180,E1 12031.434,E2 12031.434} C_VEL
LIN {X 0,Y 257.443,Z 915.922,A -85,B 0,C 180,E1 12027.326,E2 12027.326} C_VEL
LIN {X 0,Y 252.181,Z 924.635,A -85,B 0,C 180,E1 12023.206,E2 12023.206} C_VEL
LIN {X 0,Y 247.522,Z 932.58,A -85,B 0,C 180,E1 12018.348,E2 12018.348} C_VEL
LIN {X 0,Y 244.284,Z 938.5,A -85,B 0,C 180,E1 12013.434,E2 12013.434} C_VEL
LIN {X 0,Y 242.294,Z 942.602,A -85,B 0,C 180,E1 12008.537,E2 12008.537} C_VEL
LIN {X 0,Y 241.259,Z 944.991,A -85,B 0,C 180,E1 12003.727,E2 12003.727} C_VEL
LIN {X 0,Y 240.867,Z 945.873,A -85,B 0,C 180,E1 11999.05,E2 11999.05} C_VEL
LIN {X 0,Y 240.842,Z 945.463,A -85,B 0,C 180,E1 11994.522,E2 11994.522} C_VEL
LIN {X 0,Y 241.182,Z 943.596,A -85,B 0,C 180,E1 11989.867,E2 11989.867} C_VEL
LIN {X 0,Y 242.12,Z 940.166,A -85,B 0,C 180,E1 11985.074,E2 11985.074} C_VEL
LIN {X 0,Y 244.016,Z 934.932,A -85,B 0,C 180,E1 11980.143,E2 11980.143} C_VEL
LIN {X 0,Y 246.844,Z 928.354,A -85,B 0,C 180,E1 11975.574,E2 11975.574} C_VEL
LIN {X 0,Y 250.998,Z 919.519,A -85,B 0,C 180,E1 11970.893,E2 11970.893} C_VEL
LIN {X 0,Y 256.03,Z 909.203,A -85,B 0,C 180,E1 11966.637,E2 11966.637} C_VEL
LIN {X 0,Y 261.476,Z 898.11,A -85,B 0,C 180,E1 11962.967,E2 11962.967} C_VEL
LIN {X 0,Y 267.755,Z 885.042,A -85,B 0,C 180,E1 11959.452,E2 11959.452} C_VEL
LIN {X 0,Y 274.412,Z 870.553,A -85,B 0,C 180,E1 11956.296,E2 11956.296} C_VEL
LIN {X 0,Y 281.018,Z 855.176,A -85,B 0,C 180,E1 11953.565,E2 11953.565} C_VEL
LIN {X 0,Y 287.862,Z 837.581,A -85,B 0,C 180,E1 11951.045,E2 11951.045} C_VEL
LIN {X 0,Y 294.098,Z 819.616,A -85,B 0,C 180,E1 11948.978,E2 11948.978} C_VEL
LIN {X 0,Y 299.786,Z 800.838,A -85,B 0,C 180,E1 11947.235,E2 11947.235} C_VEL
LIN {X 0,Y 305.092,Z 780.01,A -85,B 0,C 180,E1 11945.71,E2 11945.71} C_VEL
LIN {X 0,Y 309.37,Z 759.173,A -85,B 0,C 180,E1 11944.545,E2 11944.545} C_VEL
LIN {X 0,Y 312.682,Z 738.026,A -85,B 0,C 180,E1 11943.677,E2 11943.677} C_VEL
LIN {X 0,Y 314.982,Z 715.868,A -85,B 0,C 180,E1 11943.056,E2 11943.056} C_VEL
LIN {X 0,Y 327.275,Z 552.283,A -85,B 0,C 180,E1 11939.448,E2 11939.448} C_VEL
LIN {X 0,Y 318.887,Z 537.458,A -85,B 0,C 180,E1 11936.435,E2 11936.435} C_VEL
LIN {X 0,Y 310.224,Z 523.671,A -85,B 0,C 180,E1 11932.972,E2 11932.972} C_VEL
LIN {X 0,Y 303.479,Z 513.626,A -85,B 0,C 180,E1 11929.932,E2 11929.932} C_VEL
LIN {X 0,Y 301.834,Z 511.223,A -85,B 0,C 180,E1 11929.133,E2 11929.133} C_VEL
LIN {X 0,Y 299.372,Z 508.68,A -85,B 0,C 180,E1 11927.938,E2 11927.938} C_VEL
LIN {X 0,Y 294.961,Z 507.148,A -85,B 0,C 180,E1 11925.855,E2 11925.855} C_VEL
LIN {X 0,Y 290.849,Z 505.606,A -85,B 0,C 180,E1 11923.702,E2 11923.702} C_VEL
LIN {X 0,Y 289.386,Z 504.017,A -85,B 0,C 180,E1 11922.802,E2 11922.802} C_VEL
LIN {X 0,Y 284.246,Z 497.275,A -85,B 0,C 180,E1 11919.155,E2 11919.155} C_VEL
LIN {X 0,Y 280.201,Z 491.948,A -85,B 0,C 180,E1 11915.693,E2 11915.693} C_VEL
LIN {X 0,Y 276.028,Z 486.697,A -85,B 0,C 180,E1 11911.198,E2 11911.198} C_VEL
LIN {X 0,Y 271.808,Z 481.402,A -85,B 0,C 180,E1 11903.869,E2 11903.869} C_VEL
LIN {X 0,Y 270.473,Z 480.305,A -85,B 0,C 180,E1 11898.091,E2 11898.091} C_VEL
LIN {X 0,Y 270.947,Z 480.704,A -85,B 0,C 180,E1 11892.576,E2 11892.576} C_VEL
LIN {X 0,Y 272.196,Z 481.928,A -85,B 0,C 180,E1 11888.824,E2 11888.824} C_VEL
LIN {X 0,Y 276.934,Z 487.662,A -85,B 0,C 180,E1 11881.449,E2 11881.449} C_VEL
LIN {X 0,Y 280.831,Z 492.482,A -85,B 0,C 180,E1 11877.45,E2 11877.45} C_VEL
LIN {X 0,Y 286.08,Z 499.316,A -85,B 0,C 180,E1 11873.176,E2 11873.176} C_VEL
LIN {X 0,Y 290.909,Z 505.755,A -85,B 0,C 180,E1 11869.905,E2 11869.905} C_VEL
LIN {X 0,Y 296.733,Z 513.589,A -85,B 0,C 180,E1 11866.507,E2 11866.507} C_VEL
LIN {X 0,Y 304.103,Z 524.173,A -85,B 0,C 180,E1 11862.788,E2 11862.788} C_VEL
LIN {X 0,Y 311.81,Z 535.836,A -85,B 0,C 180,E1 11859.395,E2 11859.395} C_VEL
LIN {X 0,Y 320.237,Z 549.49,A -85,B 0,C 180,E1 11856.102,E2 11856.102} C_VEL
LIN {X 0,Y 327.225,Z 561.799,A -85,B 0,C 180,E1 11853.617,E2 11853.617} C_VEL
LIN {X 0,Y 313.514,Z 749.643,A -85,B 0,C 180,E1 11849.582,E2 11849.582} C_VEL
LIN {X 0,Y 310.382,Z 771.851,A -85,B 0,C 180,E1 11848.89,E2 11848.89} C_VEL
LIN {X 0,Y 306.222,Z 792.771,A -85,B 0,C 180,E1 11848.001,E2 11848.001} C_VEL
LIN {X 0,Y 301.084,Z 813.61,A -85,B 0,C 180,E1 11846.814,E2 11846.814} C_VEL
LIN {X 0,Y 295.02,Z 834.181,A -85,B 0,C 180,E1 11845.294,E2 11845.294} C_VEL
LIN {X 0,Y 288.509,Z 853.014,A -85,B 0,C 180,E1 11843.521,E2 11843.521} C_VEL
LIN {X 0,Y 281.185,Z 871.903,A -85,B 0,C 180,E1 11841.312,E2 11841.312} C_VEL
LIN {X 0,Y 273.797,Z 889.3,A -85,B 0,C 180,E1 11838.793,E2 11838.793} C_VEL
LIN {X 0,Y 266.239,Z 905.84,A -85,B 0,C 180,E1 11835.837,E2 11835.837} C_VEL
LIN {X 0,Y 258.893,Z 920.982,A -85,B 0,C 180,E1 11832.469,E2 11832.469} C_VEL
LIN {X 0,Y 252.187,Z 934.478,A -85,B 0,C 180,E1 11828.792,E2 11828.792} C_VEL
LIN {X 0,Y 246.131,Z 946.834,A -85,B 0,C 180,E1 11824.666,E2 11824.666} C_VEL
LIN {X 0,Y 240.766,Z 958.293,A -85,B 0,C 180,E1 11819.895,E2 11819.895} C_VEL
LIN {X 0,Y 236.991,Z 967.174,A -85,B 0,C 180,E1 11815.226,E2 11815.226} C_VEL
LIN {X 0,Y 234.244,Z 975.079,A -85,B 0,C 180,E1 11809.972,E2 11809.972} C_VEL
LIN {X 0,Y 232.872,Z 980.884,A -85,B 0,C 180,E1 11804.934,E2 11804.934} C_VEL
LIN {X 0,Y 232.441,Z 984.742,A -85,B 0,C 180,E1 11800.163,E2 11800.163} C_VEL
LIN {X 0,Y 232.522,Z 987.27,A -85,B 0,C 180,E1 11795.433,E2 11795.433} C_VEL
LIN {X 0,Y 232.662,Z 988.212,A -85,B 0,C 180,E1 11790.99,E2 11790.99} C_VEL
LIN {X 0,Y 232.606,Z 988.019,A -85,B 0,C 180,E1 11787.049,E2 11787.049} C_VEL
LIN {X 0,Y 232.428,Z 986.606,A -85,B 0,C 180,E1 11782.591,E2 11782.591} C_VEL
LIN {X 0,Y 232.517,Z 983.674,A -85,B 0,C 180,E1 11777.842,E2 11777.842} C_VEL
LIN {X 0,Y 233.408,Z 978.872,A -85,B 0,C 180,E1 11772.557,E2 11772.557} C_VEL
LIN {X 0,Y 235.498,Z 972.35,A -85,B 0,C 180,E1 11767.278,E2 11767.278} C_VEL
LIN {X 0,Y 239.048,Z 963.891,A -85,B 0,C 180,E1 11762.072,E2 11762.072} C_VEL
LIN {X 0,Y 244.188,Z 953.498,A -85,B 0,C 180,E1 11757.011,E2 11757.011} C_VEL
LIN {X 0,Y 250.595,Z 941.593,A -85,B 0,C 180,E1 11752.385,E2 11752.385} C_VEL
LIN {X 0,Y 257.605,Z 928.978,A -85,B 0,C 180,E1 11748.424,E2 11748.424} C_VEL
LIN {X 0,Y 265.754,Z 914.125,A -85,B 0,C 180,E1 11744.685,E2 11744.685} C_VEL
LIN {X 0,Y 274.16,Z 898.266,A -85,B 0,C 180,E1 11741.465,E2 11741.465} C_VEL
LIN {X 0,Y 282.819,Z 880.955,A -85,B 0,C 180,E1 11738.629,E2 11738.629} C_VEL
LIN {X 0,Y 290.967,Z 863.419,A -85,B 0,C 180,E1 11736.32,E2 11736.32} C_VEL
LIN {X 0,Y 298.937,Z 844.197,A -85,B 0,C 180,E1 11734.305,E2 11734.305} C_VEL
LIN {X 0,Y 305.958,Z 825.091,A -85,B 0,C 180,E1 11732.711,E2 11732.711} C_VEL
LIN {X 0,Y 312.204,Z 805.476,A -85,B 0,C 180,E1 11731.417,E2 11731.417} C_VEL
LIN {X 0,Y 317.578,Z 785.165,A -85,B 0,C 180,E1 11730.394,E2 11730.394} C_VEL
LIN {X 0,Y 322.007,Z 763.859,A -85,B 0,C 180,E1 11729.599,E2 11729.599} C_VEL
LIN {X 0,Y 325.308,Z 740.523,A -85,B 0,C 180,E1 11728.948,E2 11728.948} C_VEL
LIN {X 0,Y 340.838,Z 566.127,A -85,B 0,C 180,E1 11725.173,E2 11725.173} C_VEL
LIN {X 0,Y 337.379,Z 558.576,A -85,B 0,C 180,E1 11722.936,E2 11722.936} C_VEL
LIN {X 0,Y 334.272,Z 552.166,A -85,B 0,C 180,E1 11720.485,E2 11720.485} C_VEL
LIN {X 0,Y 332.583,Z 548.954,A -85,B 0,C 180,E1 11718.855,E2 11718.855} C_VEL
LIN {X 0,Y 330.968,Z 545.778,A -85,B 0,C 180,E1 11716.858,E2 11716.858} C_VEL
LIN {X 0,Y 329.185,Z 542.106,A -85,B 0,C 180,E1 11712.989,E2 11712.989} C_VEL
LIN {X 0,Y 329.046,Z 542.048,A -85,B 0,C 180,E1 11709.267,E2 11709.267} C_VEL
LIN {X 0,Y 330.458,Z 545.405,A -85,B 0,C 180,E1 11705.527,E2 11705.527} C_VEL
LIN {X 0,Y 331.477,Z 547.488,A -85,B 0,C 180,E1 11704.064,E2 11704.064} C_VEL
LIN {X 0,Y 333.359,Z 551.215,A -85,B 0,C 180,E1 11701.976,E2 11701.976} C_VEL
LIN {X 0,Y 336.288,Z 557.47,A -85,B 0,C 180,E1 11699.446,E2 11699.446} C_VEL
LIN {X 0,Y 339.781,Z 565.129,A -85,B 0,C 180,E1 11697.048,E2 11697.048} C_VEL
LIN {X 0,Y 339.847,Z 565.9,A -85,B 0,C 180,E1 11696.964,E2 11696.964} C_VEL
LIN {X 0,Y 323.376,Z 732.816,A -85,B 0,C 180,E1 11693.27,E2 11693.27} C_VEL
LIN {X 0,Y 320.057,Z 753.552,A -85,B 0,C 180,E1 11692.559,E2 11692.559} C_VEL
LIN {X 0,Y 315.753,Z 773.441,A -85,B 0,C 180,E1 11691.624,E2 11691.624} C_VEL
LIN {X 0,Y 310.287,Z 793.625,A -85,B 0,C 180,E1 11690.382,E2 11690.382} C_VEL
LIN {X 0,Y 304.116,Z 812.497,A -85,B 0,C 180,E1 11688.9,E2 11688.9} C_VEL
LIN {X 0,Y 296.969,Z 831.014,A -85,B 0,C 180,E1 11687.061,E2 11687.061} C_VEL
LIN {X 0,Y 289.386,Z 848.237,A -85,B 0,C 180,E1 11684.928,E2 11684.928} C_VEL
LIN {X 0,Y 281.41,Z 864.49,A -85,B 0,C 180,E1 11682.421,E2 11682.421} C_VEL
LIN {X 0,Y 272.983,Z 880.141,A -85,B 0,C 180,E1 11679.413,E2 11679.413} C_VEL
LIN {X 0,Y 265.247,Z 893.499,A -85,B 0,C 180,E1 11676.212,E2 11676.212} C_VEL
LIN {X 0,Y 257.675,Z 905.893,A -85,B 0,C 180,E1 11672.499,E2 11672.499} C_VEL
LIN {X 0,Y 250.72,Z 916.784,A -85,B 0,C 180,E1 11668.346,E2 11668.346} C_VEL
LIN {X 0,Y 244.892,Z 925.834,A -85,B 0,C 180,E1 11663.929,E2 11663.929} C_VEL
LIN {X 0,Y 240.181,Z 933.321,A -85,B 0,C 180,E1 11659.187,E2 11659.187} C_VEL
LIN {X 0,Y 236.704,Z 939.181,A -85,B 0,C 180,E1 11654.176,E2 11654.176} C_VEL
LIN {X 0,Y 234.504,Z 943.315,A -85,B 0,C 180,E1 11649.104,E2 11649.104} C_VEL
LIN {X 0,Y 233.36,Z 945.698,A -85,B 0,C 180,E1 11644.137,E2 11644.137} C_VEL
LIN {X 0,Y 232.916,Z 946.596,A -85,B 0,C 180,E1 11639.293,E2 11639.293} C_VEL
LIN {X 0,Y 232.875,Z 946.163,A -85,B 0,C 180,E1 11634.461,E2 11634.461} C_VEL
LIN {X 0,Y 233.223,Z 944.347,A -85,B 0,C 180,E1 11629.79,E2 11629.79} C_VEL
LIN {X 0,Y 234.214,Z 940.942,A -85,B 0,C 180,E1 11624.835,E2 11624.835} C_VEL
LIN {X 0,Y 236.096,Z 936.051,A -85,B 0,C 180,E1 11619.994,E2 11619.994} C_VEL
LIN {X 0,Y 239.024,Z 929.586,A -85,B 0,C 180,E1 11615.275,E2 11615.275} C_VEL
LIN {X 0,Y 243.061,Z 921.333,A -85,B 0,C 180,E1 11610.702,E2 11610.702} C_VEL
LIN {X 0,Y 248.237,Z 911.23,A -85,B 0,C 180,E1 11606.3,E2 11606.3} C_VEL
LIN {X 0,Y 254.292,Z 899.507,A -85,B 0,C 180,E1 11602.246,E2 11602.246} C_VEL
LIN {X 0,Y 260.687,Z 886.823,A -85,B 0,C 180,E1 11598.715,E2 11598.715} C_VEL
LIN {X 0,Y 267.565,Z 872.55,A -85,B 0,C 180,E1 11595.496,E2 11595.496} C_VEL
LIN {X 0,Y 274.863,Z 856.205,A -85,B 0,C 180,E1 11592.532,E2 11592.532} C_VEL
LIN {X 0,Y 281.68,Z 839.336,A -85,B 0,C 180,E1 11590.073,E2 11590.073} C_VEL
LIN {X 0,Y 288.115,Z 821.61,A -85,B 0,C 180,E1 11587.984,E2 11587.984} C_VEL
LIN {X 0,Y 294.261,Z 802.159,A -85,B 0,C 180,E1 11586.146,E2 11586.146} C_VEL
LIN {X 0,Y 299.443,Z 782.755,A -85,B 0,C 180,E1 11584.694,E2 11584.694} C_VEL
LIN {X 0,Y 303.919,Z 762.227,A -85,B 0,C 180,E1 11583.503,E2 11583.503} C_VEL
LIN {X 0,Y 307.582,Z 740.11,A -85,B 0,C 180,E1 11582.564,E2 11582.564} C_VEL
LIN {X 0,Y 310.044,Z 717.653,A -85,B 0,C 180,E1 11581.921,E2 11581.921} C_VEL
LIN {X 0,Y 322.632,Z 556.2,A -85,B 0,C 180,E1 11578.361,E2 11578.361} C_VEL
LIN {X 0,Y 314.458,Z 541.741,A -85,B 0,C 180,E1 11575.28,E2 11575.28} C_VEL
LIN {X 0,Y 305.923,Z 527.914,A -85,B 0,C 180,E1 11571.666,E2 11571.666} C_VEL
LIN {X 0,Y 298.348,Z 516.614,A -85,B 0,C 180,E1 11567.994,E2 11567.994} C_VEL
LIN {X 0,Y 292.012,Z 507.633,A -85,B 0,C 180,E1 11564.445,E2 11564.445} C_VEL
LIN {X 0,Y 289.386,Z 504.017,A -85,B 0,C 180,E1 11562.802,E2 11562.802} C_VEL
LIN {X 0,Y 287.497,Z 502.271,A -85,B 0,C 180,E1 11561.587,E2 11561.587} C_VEL
LIN {X 0,Y 284.21,Z 501.944,A -85,B 0,C 180,E1 11559.559,E2 11559.559} C_VEL
LIN {X 0,Y 280.726,Z 501.796,A -85,B 0,C 180,E1 11557.147,E2 11557.147} C_VEL
LIN {X 0,Y 279.355,Z 500.413,A -85,B 0,C 180,E1 11555.956,E2 11555.956} C_VEL
LIN {X 0,Y 274.599,Z 494.36,A -85,B 0,C 180,E1 11550.755,E2 11550.755} C_VEL
LIN {X 0,Y 270.593,Z 489.232,A -85,B 0,C 180,E1 11543.521,E2 11543.521} C_VEL
LIN {X 0,Y 269.396,Z 488.23,A -85,B 0,C 180,E1 11537.719,E2 11537.719} C_VEL
LIN {X 0,Y 269.918,Z 488.68,A -85,B 0,C 180,E1 11532.407,E2 11532.407} C_VEL
LIN {X 0,Y 271.091,Z 489.873,A -85,B 0,C 180,E1 11528.912,E2 11528.912} C_VEL
LIN {X 0,Y 275.647,Z 495.554,A -85,B 0,C 180,E1 11521.663,E2 11521.663} C_VEL
LIN {X 0,Y 280.047,Z 501.191,A -85,B 0,C 180,E1 11517.135,E2 11517.135} C_VEL
LIN {X 0,Y 284.437,Z 506.983,A -85,B 0,C 180,E1 11513.542,E2 11513.542} C_VEL
LIN {X 0,Y 289.094,Z 513.293,A -85,B 0,C 180,E1 11510.313,E2 11510.313} C_VEL
LIN {X 0,Y 294.779,Z 521.152,A -85,B 0,C 180,E1 11506.915,E2 11506.915} C_VEL
LIN {X 0,Y 301.768,Z 531.37,A -85,B 0,C 180,E1 11503.296,E2 11503.296} C_VEL
LIN {X 0,Y 309.055,Z 542.621,A -85,B 0,C 180,E1 11499.994,E2 11499.994} C_VEL
LIN {X 0,Y 317.127,Z 555.948,A -85,B 0,C 180,E1 11496.741,E2 11496.741} C_VEL
LIN {X 0,Y 322.578,Z 565.832,A -85,B 0,C 180,E1 11494.721,E2 11494.721} C_VEL
LIN {X 0,Y 308.724,Z 749.176,A -85,B 0,C 180,E1 11490.77,E2 11490.77} C_VEL
LIN {X 0,Y 305.535,Z 771.288,A -85,B 0,C 180,E1 11490.082,E2 11490.082} C_VEL
LIN {X 0,Y 301.412,Z 791.63,A -85,B 0,C 180,E1 11489.228,E2 11489.228} C_VEL
LIN {X 0,Y 296.277,Z 812.147,A -85,B 0,C 180,E1 11488.08,E2 11488.08} C_VEL
LIN {X 0,Y 290.315,Z 831.942,A -85,B 0,C 180,E1 11486.639,E2 11486.639} C_VEL
LIN {X 0,Y 283.618,Z 851.035,A -85,B 0,C 180,E1 11484.879,E2 11484.879} C_VEL
LIN {X 0,Y 276.038,Z 870.188,A -85,B 0,C 180,E1 11482.667,E2 11482.667} C_VEL
LIN {X 0,Y 268.379,Z 887.708,A -85,B 0,C 180,E1 11480.15,E2 11480.15} C_VEL
LIN {X 0,Y 260.452,Z 904.387,A -85,B 0,C 180,E1 11477.163,E2 11477.163} C_VEL
LIN {X 0,Y 252.838,Z 919.521,A -85,B 0,C 180,E1 11473.797,E2 11473.797} C_VEL
LIN {X 0,Y 245.304,Z 934.058,A -85,B 0,C 180,E1 11469.792,E2 11469.792} C_VEL
LIN {X 0,Y 238.955,Z 946.38,A -85,B 0,C 180,E1 11465.569,E2 11465.569} C_VEL
LIN {X 0,Y 233.549,Z 957.273,A -85,B 0,C 180,E1 11460.918,E2 11460.918} C_VEL
LIN {X 0,Y 229.307,Z 966.663,A -85,B 0,C 180,E1 11455.856,E2 11455.856} C_VEL
LIN {X 0,Y 226.388,Z 974.534,A -85,B 0,C 180,E1 11450.426,E2 11450.426} C_VEL
LIN {X 0,Y 224.92,Z 980.299,A -85,B 0,C 180,E1 11445.21,E2 11445.21} C_VEL
LIN {X 0,Y 224.458,Z 984.223,A -85,B 0,C 180,E1 11440.12,E2 11440.12} C_VEL
LIN {X 0,Y 224.552,Z 986.598,A -85,B 0,C 180,E1 11435.371,E2 11435.371} C_VEL
LIN {X 0,Y 224.694,Z 987.486,A -85,B 0,C 180,E1 11431.025,E2 11431.025} C_VEL
LIN {X 0,Y 224.633,Z 987.303,A -85,B 0,C 180,E1 11426.944,E2 11426.944} C_VEL
LIN {X 0,Y 224.445,Z 985.911,A -85,B 0,C 180,E1 11422.326,E2 11422.326} C_VEL
LIN {X 0,Y 224.558,Z 982.987,A -85,B 0,C 180,E1 11417.404,E2 11417.404} C_VEL
LIN {X 0,Y 225.565,Z 978.207,A -85,B 0,C 180,E1 11411.93,E2 11411.93} C_VEL
LIN {X 0,Y 227.867,Z 971.694,A -85,B 0,C 180,E1 11406.472,E2 11406.472} C_VEL
LIN {X 0,Y 231.646,Z 963.413,A -85,B 0,C 180,E1 11401.187,E2 11401.187} C_VEL
LIN {X 0,Y 237.221,Z 952.924,A -85,B 0,C 180,E1 11395.912,E2 11395.912} C_VEL
LIN {X 0,Y 243.664,Z 941.74,A -85,B 0,C 180,E1 11391.419,E2 11391.419} C_VEL
LIN {X 0,Y 251.439,Z 928.507,A -85,B 0,C 180,E1 11387.165,E2 11387.165} C_VEL
LIN {X 0,Y 259.488,Z 914.595,A -85,B 0,C 180,E1 11383.59,E2 11383.59} C_VEL
LIN {X 0,Y 268.772,Z 897.979,A -85,B 0,C 180,E1 11380.148,E2 11380.148} C_VEL
LIN {X 0,Y 277.481,Z 881.387,A -85,B 0,C 180,E1 11377.398,E2 11377.398} C_VEL
LIN {X 0,Y 286.225,Z 863.346,A -85,B 0,C 180,E1 11375.008,E2 11375.008} C_VEL
LIN {X 0,Y 294.237,Z 844.825,A -85,B 0,C 180,E1 11373.057,E2 11373.057} C_VEL
LIN {X 0,Y 302.043,Z 824.398,A -85,B 0,C 180,E1 11371.355,E2 11371.355} C_VEL
LIN {X 0,Y 308.482,Z 804.878,A -85,B 0,C 180,E1 11370.082,E2 11370.082} C_VEL
LIN {X 0,Y 313.836,Z 785.297,A -85,B 0,C 180,E1 11369.106,E2 11369.106} C_VEL
LIN {X 0,Y 318.472,Z 763.77,A -85,B 0,C 180,E1 11368.308,E2 11368.308} C_VEL
LIN {X 0,Y 321.91,Z 740.565,A -85,B 0,C 180,E1 11367.662,E2 11367.662} C_VEL
LIN {X 0,Y 337.719,Z 570.765,A -85,B 0,C 180,E1 11363.998,E2 11363.998} C_VEL
LIN {X 0,Y 334.121,Z 562.759,A -85,B 0,C 180,E1 11361.366,E2 11361.366} C_VEL
LIN {X 0,Y 331.446,Z 557.067,A -85,B 0,C 180,E1 11358.831,E2 11358.831} C_VEL
LIN {X 0,Y 329.667,Z 553.51,A -85,B 0,C 180,E1 11356.564,E2 11356.564} C_VEL
LIN {X 0,Y 328.06,Z 549.979,A -85,B 0,C 180,E1 11352.788,E2 11352.788} C_VEL
LIN {X 0,Y 328.012,Z 550.041,A -85,B 0,C 180,E1 11349.057,E2 11349.057} C_VEL
LIN {X 0,Y 329.721,Z 554.195,A -85,B 0,C 180,E1 11344.957,E2 11344.957} C_VEL
LIN {X 0,Y 331.764,Z 558.624,A -85,B 0,C 180,E1 11342.418,E2 11342.418} C_VEL
LIN {X 0,Y 334.473,Z 564.771,A -85,B 0,C 180,E1 11339.914,E2 11339.914} C_VEL
LIN {X 0,Y 336.802,Z 570.272,A -85,B 0,C 180,E1 11338.157,E2 11338.157} C_VEL
LIN {X 0,Y 320.132,Z 733.191,A -85,B 0,C 180,E1 11334.572,E2 11334.572} C_VEL
LIN {X 0,Y 316.658,Z 754.235,A -85,B 0,C 180,E1 11333.857,E2 11333.857} C_VEL
LIN {X 0,Y 312.289,Z 773.851,A -85,B 0,C 180,E1 11332.946,E2 11332.946} C_VEL
LIN {X 0,Y 306.81,Z 793.472,A -85,B 0,C 180,E1 11331.755,E2 11331.755} C_VEL
LIN {X 0,Y 300.682,Z 811.684,A -85,B 0,C 180,E1 11330.351,E2 11330.351} C_VEL
LIN {X 0,Y 293.554,Z 829.703,A -85,B 0,C 180,E1 11328.606,E2 11328.606} C_VEL
LIN {X 0,Y 285.789,Z 846.908,A -85,B 0,C 180,E1 11326.533,E2 11326.533} C_VEL
LIN {X 0,Y 277.571,Z 863.218,A -85,B 0,C 180,E1 11324.086,E2 11324.086} C_VEL
LIN {X 0,Y 269.197,Z 878.346,A -85,B 0,C 180,E1 11321.266,E2 11321.266} C_VEL
LIN {X 0,Y 260.541,Z 892.667,A -85,B 0,C 180,E1 11317.908,E2 11317.908} C_VEL
LIN {X 0,Y 252.82,Z 904.645,A -85,B 0,C 180,E1 11314.367,E2 11314.367} C_VEL
LIN {X 0,Y 245.338,Z 915.776,A -85,B 0,C 180,E1 11310.222,E2 11310.222} C_VEL
LIN {X 0,Y 238.696,Z 925.502,A -85,B 0,C 180,E1 11305.563,E2 11305.563} C_VEL
LIN {X 0,Y 233.412,Z 933.31,A -85,B 0,C 180,E1 11300.655,E2 11300.655} C_VEL
LIN {X 0,Y 229.464,Z 939.443,A -85,B 0,C 180,E1 11295.449,E2 11295.449} C_VEL
LIN {X 0,Y 226.855,Z 943.812,A -85,B 0,C 180,E1 11290.044,E2 11290.044} C_VEL
LIN {X 0,Y 225.519,Z 946.297,A -85,B 0,C 180,E1 11284.877,E2 11284.877} C_VEL
LIN {X 0,Y 224.975,Z 947.315,A -85,B 0,C 180,E1 11279.845,E2 11279.845} C_VEL
LIN {X 0,Y 224.892,Z 947.007,A -85,B 0,C 180,E1 11274.977,E2 11274.977} C_VEL
LIN {X 0,Y 225.189,Z 945.353,A -85,B 0,C 180,E1 11270.256,E2 11270.256} C_VEL
LIN {X 0,Y 226.167,Z 942.15,A -85,B 0,C 180,E1 11265.113,E2 11265.113} C_VEL
LIN {X 0,Y 228.049,Z 937.466,A -85,B 0,C 180,E1 11260.095,E2 11260.095} C_VEL
LIN {X 0,Y 231.2,Z 930.749,A -85,B 0,C 180,E1 11254.956,E2 11254.956} C_VEL
LIN {X 0,Y 235.391,Z 922.627,A -85,B 0,C 180,E1 11250.238,E2 11250.238} C_VEL
LIN {X 0,Y 240.763,Z 912.667,A -85,B 0,C 180,E1 11245.708,E2 11245.708} C_VEL
LIN {X 0,Y 246.931,Z 901.312,A -85,B 0,C 180,E1 11241.613,E2 11241.613} C_VEL
LIN {X 0,Y 253.664,Z 888.604,A -85,B 0,C 180,E1 11237.937,E2 11237.937} C_VEL
LIN {X 0,Y 260.76,Z 874.463,A -85,B 0,C 180,E1 11234.654,E2 11234.654} C_VEL
LIN {X 0,Y 268.034,Z 858.85,A -85,B 0,C 180,E1 11231.735,E2 11231.735} C_VEL
LIN {X 0,Y 275.038,Z 842.363,A -85,B 0,C 180,E1 11229.236,E2 11229.236} C_VEL
LIN {X 0,Y 282.212,Z 823.521,A -85,B 0,C 180,E1 11226.949,E2 11226.949} C_VEL
LIN {X 0,Y 288.543,Z 804.371,A -85,B 0,C 180,E1 11225.097,E2 11225.097} C_VEL
LIN {X 0,Y 293.887,Z 785.406,A -85,B 0,C 180,E1 11223.638,E2 11223.638} C_VEL
LIN {X 0,Y 298.728,Z 764.167,A -85,B 0,C 180,E1 11222.379,E2 11222.379} C_VEL
LIN {X 0,Y 302.48,Z 742.527,A -85,B 0,C 180,E1 11221.437,E2 11221.437} C_VEL
LIN {X 0,Y 305.038,Z 721.103,A -85,B 0,C 180,E1 11220.795,E2 11220.795} C_VEL
LIN {X 0,Y 318.063,Z 560.076,A -85,B 0,C 180,E1 11217.225,E2 11217.225} C_VEL
LIN {X 0,Y 310.503,Z 546.703,A -85,B 0,C 180,E1 11214.241,E2 11214.241} C_VEL
LIN {X 0,Y 302.78,Z 533.956,A -85,B 0,C 180,E1 11210.825,E2 11210.825} C_VEL
LIN {X 0,Y 295.613,Z 523.164,A -85,B 0,C 180,E1 11207.221,E2 11207.221} C_VEL
LIN {X 0,Y 289.978,Z 514.942,A -85,B 0,C 180,E1 11203.942,E2 11203.942} C_VEL
LIN {X 0,Y 286.054,Z 509.621,A -85,B 0,C 180,E1 11201.348,E2 11201.348} C_VEL
LIN {X 0,Y 282.611,Z 504.879,A -85,B 0,C 180,E1 11198.772,E2 11198.772} C_VEL
LIN {X 0,Y 279.355,Z 500.413,A -85,B 0,C 180,E1 11195.956,E2 11195.956} C_VEL
LIN {X 0,Y 277.958,Z 499.106,A -85,B 0,C 180,E1 11194.653,E2 11194.653} C_VEL
LIN {X 0,Y 275.779,Z 499.556,A -85,B 0,C 180,E1 11192.742,E2 11192.742} C_VEL
LIN {X 0,Y 272.792,Z 501.186,A -85,B 0,C 180,E1 11189.738,E2 11189.738} C_VEL
LIN {X 0,Y 272.018,Z 500.839,A -85,B 0,C 180,E1 11188.682,E2 11188.682} C_VEL
LIN {X 0,Y 269.468,Z 497.132,A -85,B 0,C 180,E1 11183.393,E2 11183.393} C_VEL
LIN {X 0,Y 268.331,Z 496.159,A -85,B 0,C 180,E1 11177.792,E2 11177.792} C_VEL
LIN {X 0,Y 268.835,Z 496.603,A -85,B 0,C 180,E1 11172.458,E2 11172.458} C_VEL
LIN {X 0,Y 269.92,Z 497.696,A -85,B 0,C 180,E1 11169.166,E2 11169.166} C_VEL
LIN {X 0,Y 274.283,Z 503.299,A -85,B 0,C 180,E1 11161.985,E2 11161.985} C_VEL
LIN {X 0,Y 278.505,Z 508.815,A -85,B 0,C 180,E1 11157.531,E2 11157.531} C_VEL
LIN {X 0,Y 282.741,Z 514.543,A -85,B 0,C 180,E1 11153.962,E2 11153.962} C_VEL
LIN {X 0,Y 287.193,Z 520.695,A -85,B 0,C 180,E1 11150.785,E2 11150.785} C_VEL
LIN {X 0,Y 292.674,Z 528.444,A -85,B 0,C 180,E1 11147.421,E2 11147.421} C_VEL
LIN {X 0,Y 299.365,Z 538.42,A -85,B 0,C 180,E1 11143.857,E2 11143.857} C_VEL
LIN {X 0,Y 306.327,Z 549.404,A -85,B 0,C 180,E1 11140.603,E2 11140.603} C_VEL
LIN {X 0,Y 314.362,Z 562.935,A -85,B 0,C 180,E1 11137.267,E2 11137.267} C_VEL
LIN {X 0,Y 318.022,Z 569.702,A -85,B 0,C 180,E1 11135.854,E2 11135.854} C_VEL
LIN {X 0,Y 304.064,Z 748.765,A -85,B 0,C 180,E1 11131.993,E2 11131.993} C_VEL
LIN {X 0,Y 300.791,Z 770.907,A -85,B 0,C 180,E1 11131.305,E2 11131.305} C_VEL
LIN {X 0,Y 296.331,Z 792.221,A -85,B 0,C 180,E1 11130.408,E2 11130.408} C_VEL
LIN {X 0,Y 290.927,Z 812.954,A -85,B 0,C 180,E1 11129.232,E2 11129.232} C_VEL
LIN {X 0,Y 284.501,Z 833.538,A -85,B 0,C 180,E1 11127.711,E2 11127.711} C_VEL
LIN {X 0,Y 277.296,Z 853.149,A -85,B 0,C 180,E1 11125.85,E2 11125.85} C_VEL
LIN {X 0,Y 269.824,Z 871.164,A -85,B 0,C 180,E1 11123.709,E2 11123.709} C_VEL
LIN {X 0,Y 261.912,Z 888.524,A -85,B 0,C 180,E1 11121.154,E2 11121.154} C_VEL
LIN {X 0,Y 253.775,Z 905.042,A -85,B 0,C 180,E1 11118.134,E2 11118.134} C_VEL
LIN {X 0,Y 245.902,Z 919.976,A -85,B 0,C 180,E1 11114.708,E2 11114.708} C_VEL
LIN {X 0,Y 238.501,Z 933.593,A -85,B 0,C 180,E1 11110.848,E2 11110.848} C_VEL
LIN {X 0,Y 231.841,Z 945.898,A -85,B 0,C 180,E1 11106.529,E2 11106.529} C_VEL
LIN {X 0,Y 226.143,Z 956.792,A -85,B 0,C 180,E1 11101.75,E2 11101.75} C_VEL
LIN {X 0,Y 221.839,Z 965.713,A -85,B 0,C 180,E1 11096.795,E2 11096.795} C_VEL
LIN {X 0,Y 218.632,Z 973.744,A -85,B 0,C 180,E1 11091.103,E2 11091.103} C_VEL
LIN {X 0,Y 216.994,Z 979.594,A -85,B 0,C 180,E1 11085.633,E2 11085.633} C_VEL
LIN {X 0,Y 216.486,Z 983.527,A -85,B 0,C 180,E1 11080.344,E2 11080.344} C_VEL
LIN {X 0,Y 216.584,Z 985.923,A -85,B 0,C 180,E1 11075.303,E2 11075.303} C_VEL
LIN {X 0,Y 216.727,Z 986.775,A -85,B 0,C 180,E1 11070.799,E2 11070.799} C_VEL
LIN {X 0,Y 216.659,Z 986.59,A -85,B 0,C 180,E1 11066.831,E2 11066.831} C_VEL
LIN {X 0,Y 216.464,Z 985.223,A -85,B 0,C 180,E1 11062.041,E2 11062.041} C_VEL
LIN {X 0,Y 216.609,Z 982.273,A -85,B 0,C 180,E1 11056.894,E2 11056.894} C_VEL
LIN {X 0,Y 217.746,Z 977.548,A -85,B 0,C 180,E1 11051.257,E2 11051.257} C_VEL
LIN {X 0,Y 220.28,Z 971.051,A -85,B 0,C 180,E1 11045.61,E2 11045.61} C_VEL
LIN {X 0,Y 224.449,Z 962.672,A -85,B 0,C 180,E1 11040.078,E2 11040.078} C_VEL
LIN {X 0,Y 230.492,Z 952.134,A -85,B 0,C 180,E1 11034.639,E2 11034.639} C_VEL
LIN {X 0,Y 237.596,Z 940.593,A -85,B 0,C 180,E1 11029.928,E2 11029.928} C_VEL
LIN {X 0,Y 245.88,Z 927.331,A -85,B 0,C 180,E1 11025.628,E2 11025.628} C_VEL
LIN {X 0,Y 254.94,Z 912.46,A -85,B 0,C 180,E1 11021.814,E2 11021.814} C_VEL
LIN {X 0,Y 264.119,Z 896.689,A -85,B 0,C 180,E1 11018.59,E2 11018.59} C_VEL
LIN {X 0,Y 273.362,Z 879.791,A -85,B 0,C 180,E1 11015.818,E2 11015.818} C_VEL
LIN {X 0,Y 282.313,Z 861.969,A -85,B 0,C 180,E1 11013.492,E2 11013.492} C_VEL
LIN {X 0,Y 290.493,Z 843.683,A -85,B 0,C 180,E1 11011.594,E2 11011.594} C_VEL
LIN {X 0,Y 298.381,Z 823.665,A -85,B 0,C 180,E1 11009.953,E2 11009.953} C_VEL
LIN {X 0,Y 304.938,Z 804.391,A -85,B 0,C 180,E1 11008.717,E2 11008.717} C_VEL
LIN {X 0,Y 310.462,Z 784.857,A -85,B 0,C 180,E1 11007.759,E2 11007.759} C_VEL
LIN {X 0,Y 315.251,Z 763.351,A -85,B 0,C 180,E1 11006.972,E2 11006.972} C_VEL
LIN {X 0,Y 318.748,Z 740.572,A -85,B 0,C 180,E1 11006.343,E2 11006.343} C_VEL
LIN {X 0,Y 334.763,Z 575.664,A -85,B 0,C 180,E1 11002.801,E2 11002.801} C_VEL
LIN {X 0,Y 331.729,Z 568.567,A -85,B 0,C 180,E1 11000.28,E2 11000.28} C_VEL
LIN {X 0,Y 329.756,Z 564.237,A -85,B 0,C 180,E1 10998.198,E2 10998.198} C_VEL
LIN {X 0,Y 328.375,Z 561.243,A -85,B 0,C 180,E1 10996.267,E2 10996.267} C_VEL
LIN {X 0,Y 326.967,Z 557.896,A -85,B 0,C 180,E1 10992.719,E2 10992.719} C_VEL
LIN {X 0,Y 326.906,Z 557.949,A -85,B 0,C 180,E1 10989.151,E2 10989.151} C_VEL
LIN {X 0,Y 328.408,Z 561.934,A -85,B 0,C 180,E1 10985.24,E2 10985.24} C_VEL
LIN {X 0,Y 330.299,Z 566.292,A -85,B 0,C 180,E1 10982.74,E2 10982.74} C_VEL
LIN {X 0,Y 332.794,Z 572.308,A -85,B 0,C 180,E1 10980.301,E2 10980.301} C_VEL
LIN {X 0,Y 333.887,Z 575.299,A -85,B 0,C 180,E1 10979.361,E2 10979.361} C_VEL
LIN {X 0,Y 317.083,Z 734.023,A -85,B 0,C 180,E1 10975.894,E2 10975.894} C_VEL
LIN {X 0,Y 313.527,Z 754.814,A -85,B 0,C 180,E1 10975.194,E2 10975.194} C_VEL
LIN {X 0,Y 308.916,Z 774.749,A -85,B 0,C 180,E1 10974.275,E2 10974.275} C_VEL
LIN {X 0,Y 303.138,Z 794.591,A -85,B 0,C 180,E1 10973.075,E2 10973.075} C_VEL
LIN {X 0,Y 296.459,Z 813.685,A -85,B 0,C 180,E1 10971.602,E2 10971.602} C_VEL
LIN {X 0,Y 288.974,Z 831.742,A -85,B 0,C 180,E1 10969.836,E2 10969.836} C_VEL
LIN {X 0,Y 280.835,Z 848.883,A -85,B 0,C 180,E1 10967.74,E2 10967.74} C_VEL
LIN {X 0,Y 271.975,Z 865.585,A -85,B 0,C 180,E1 10965.184,E2 10965.184} C_VEL
LIN {X 0,Y 263.183,Z 880.573,A -85,B 0,C 180,E1 10962.306,E2 10962.306} C_VEL
LIN {X 0,Y 254.597,Z 894.127,A -85,B 0,C 180,E1 10959.06,E2 10959.06} C_VEL
LIN {X 0,Y 245.78,Z 907.073,A -85,B 0,C 180,E1 10955.104,E2 10955.104} C_VEL
LIN {X 0,Y 238.048,Z 917.866,A -85,B 0,C 180,E1 10950.872,E2 10950.872} C_VEL
LIN {X 0,Y 231.583,Z 926.694,A -85,B 0,C 180,E1 10946.425,E2 10946.425} C_VEL
LIN {X 0,Y 226.029,Z 934.355,A -85,B 0,C 180,E1 10941.41,E2 10941.41} C_VEL
LIN {X 0,Y 221.878,Z 940.306,A -85,B 0,C 180,E1 10936.128,E2 10936.128} C_VEL
LIN {X 0,Y 219.132,Z 944.519,A -85,B 0,C 180,E1 10930.72,E2 10930.72} C_VEL
LIN {X 0,Y 217.64,Z 947.015,A -85,B 0,C 180,E1 10925.362,E2 10925.362} C_VEL
LIN {X 0,Y 217.015,Z 948.046,A -85,B 0,C 180,E1 10919.981,E2 10919.981} C_VEL
LIN {X 0,Y 216.92,Z 947.736,A -85,B 0,C 180,E1 10915.084,E2 10915.084} C_VEL
LIN {X 0,Y 217.237,Z 946.069,A -85,B 0,C 180,E1 10910.124,E2 10910.124} C_VEL
LIN {X 0,Y 218.263,Z 942.911,A -85,B 0,C 180,E1 10904.85,E2 10904.85} C_VEL
LIN {X 0,Y 220.389,Z 937.949,A -85,B 0,C 180,E1 10899.394,E2 10899.394} C_VEL
LIN {X 0,Y 223.789,Z 931.185,A -85,B 0,C 180,E1 10894.094,E2 10894.094} C_VEL
LIN {X 0,Y 228.268,Z 922.983,A -85,B 0,C 180,E1 10889.242,E2 10889.242} C_VEL
LIN {X 0,Y 233.971,Z 912.934,A -85,B 0,C 180,E1 10884.6,E2 10884.6} C_VEL
LIN {X 0,Y 240.872,Z 900.772,A -85,B 0,C 180,E1 10880.196,E2 10880.196} C_VEL
LIN {X 0,Y 247.986,Z 887.809,A -85,B 0,C 180,E1 10876.471,E2 10876.471} C_VEL
LIN {X 0,Y 255.469,Z 873.451,A -85,B 0,C 180,E1 10873.16,E2 10873.16} C_VEL
LIN {X 0,Y 263.354,Z 857.032,A -85,B 0,C 180,E1 10870.131,E2 10870.131} C_VEL
LIN {X 0,Y 270.69,Z 840.063,A -85,B 0,C 180,E1 10867.634,E2 10867.634} C_VEL
LIN {X 0,Y 277.574,Z 822.225,A -85,B 0,C 180,E1 10865.524,E2 10865.524} C_VEL
LIN {X 0,Y 284.127,Z 802.657,A -85,B 0,C 180,E1 10863.675,E2 10863.675} C_VEL
LIN {X 0,Y 289.638,Z 783.106,A -85,B 0,C 180,E1 10862.219,E2 10862.219} C_VEL
LIN {X 0,Y 294.335,Z 762.639,A -85,B 0,C 180,E1 10861.043,E2 10861.043} C_VEL
LIN {X 0,Y 298.17,Z 740.688,A -85,B 0,C 180,E1 10860.117,E2 10860.117} C_VEL
LIN {X 0,Y 300.78,Z 718.118,A -85,B 0,C 180,E1 10859.474,E2 10859.474} C_VEL
LIN {X 0,Y 313.524,Z 563.994,A -85,B 0,C 180,E1 10856.056,E2 10856.056} C_VEL
LIN {X 0,Y 306.611,Z 551.616,A -85,B 0,C 180,E1 10853.186,E2 10853.186} C_VEL
LIN {X 0,Y 299.252,Z 539.415,A -85,B 0,C 180,E1 10849.771,E2 10849.771} C_VEL
LIN {X 0,Y 292.639,Z 529.276,A -85,B 0,C 180,E1 10846.273,E2 10846.273} C_VEL
LIN {X 0,Y 287.791,Z 522.039,A -85,B 0,C 180,E1 10843.328,E2 10843.328} C_VEL
LIN {X 0,Y 284.136,Z 516.97,A -85,B 0,C 180,E1 10840.833,E2 10840.833} C_VEL
LIN {X 0,Y 280.848,Z 512.337,A -85,B 0,C 180,E1 10838.278,E2 10838.278} C_VEL
LIN {X 0,Y 277.115,Z 507.207,A -85,B 0,C 180,E1 10834.882,E2 10834.882} C_VEL
LIN {X 0,Y 273.349,Z 502.207,A -85,B 0,C 180,E1 10830.56,E2 10830.56} C_VEL
LIN {X 0,Y 272.018,Z 500.839,A -85,B 0,C 180,E1 10828.682,E2 10828.682} C_VEL
LIN {X 0,Y 270.942,Z 500.618,A -85,B 0,C 180,E1 10827.056,E2 10827.056} C_VEL
LIN {X 0,Y 268.828,Z 503.306,A -85,B 0,C 180,E1 10823.796,E2 10823.796} C_VEL
LIN {X 0,Y 267.869,Z 504.517,A -85,B 0,C 180,E1 10821.657,E2 10821.657} C_VEL
LIN {X 0,Y 267.731,Z 504.485,A -85,B 0,C 180,E1 10821.177,E2 10821.177} C_VEL
LIN {X 0,Y 267.336,Z 504.104,A -85,B 0,C 180,E1 10814.956,E2 10814.956} C_VEL
LIN {X 0,Y 268.7,Z 505.423,A -85,B 0,C 180,E1 10809.552,E2 10809.552} C_VEL
LIN {X 0,Y 272.928,Z 511.043,A -85,B 0,C 180,E1 10802.31,E2 10802.31} C_VEL
LIN {X 0,Y 276.949,Z 516.431,A -85,B 0,C 180,E1 10797.932,E2 10797.932} C_VEL
LIN {X 0,Y 281.03,Z 522.09,A -85,B 0,C 180,E1 10794.386,E2 10794.386} C_VEL
LIN {X 0,Y 285.279,Z 528.078,A -85,B 0,C 180,E1 10791.269,E2 10791.269} C_VEL
LIN {X 0,Y 290.636,Z 535.85,A -85,B 0,C 180,E1 10787.887,E2 10787.887} C_VEL
LIN {X 0,Y 297.053,Z 545.606,A -85,B 0,C 180,E1 10784.379,E2 10784.379} C_VEL
LIN {X 0,Y 303.708,Z 556.348,A -85,B 0,C 180,E1 10781.178,E2 10781.178} C_VEL
LIN {X 0,Y 311.411,Z 569.577,A -85,B 0,C 180,E1 10777.886,E2 10777.886} C_VEL
LIN {X 0,Y 313.545,Z 573.844,A -85,B 0,C 180,E1 10777.011,E2 10777.011} C_VEL
LIN {X 0,Y 299.477,Z 748.461,A -85,B 0,C 180,E1 10773.243,E2 10773.243} C_VEL
LIN {X 0,Y 296.115,Z 770.676,A -85,B 0,C 180,E1 10772.555,E2 10772.555} C_VEL
LIN {X 0,Y 291.682,Z 791.396,A -85,B 0,C 180,E1 10771.691,E2 10771.691} C_VEL
LIN {X 0,Y 286.051,Z 812.515,A -85,B 0,C 180,E1 10770.505,E2 10770.505} C_VEL
LIN {X 0,Y 279.771,Z 832.185,A -85,B 0,C 180,E1 10769.067,E2 10769.067} C_VEL
LIN {X 0,Y 272.619,Z 851.219,A -85,B 0,C 180,E1 10767.287,E2 10767.287} C_VEL
LIN {X 0,Y 264.643,Z 870.029,A -85,B 0,C 180,E1 10765.076,E2 10765.076} C_VEL
LIN {X 0,Y 256.587,Z 887.19,A -85,B 0,C 180,E1 10762.563,E2 10762.563} C_VEL
LIN {X 0,Y 247.995,Z 904.015,A -85,B 0,C 180,E1 10759.48,E2 10759.48} C_VEL
LIN {X 0,Y 239.993,Z 918.624,A -85,B 0,C 180,E1 10756.122,E2 10756.122} C_VEL
LIN {X 0,Y 232.214,Z 932.391,A -85,B 0,C 180,E1 10752.204,E2 10752.204} C_VEL
LIN {X 0,Y 225.066,Z 944.929,A -85,B 0,C 180,E1 10747.744,E2 10747.744} C_VEL
LIN {X 0,Y 219.018,Z 955.814,A -85,B 0,C 180,E1 10742.862,E2 10742.862} C_VEL
LIN {X 0,Y 214.23,Z 965.166,A -85,B 0,C 180,E1 10737.531,E2 10737.531} C_VEL
LIN {X 0,Y 210.808,Z 973.188,A -85,B 0,C 180,E1 10731.626,E2 10731.626} C_VEL
LIN {X 0,Y 209.061,Z 978.96,A -85,B 0,C 180,E1 10725.994,E2 10725.994} C_VEL
LIN {X 0,Y 208.51,Z 982.874,A -85,B 0,C 180,E1 10720.505,E2 10720.505} C_VEL
LIN {X 0,Y 208.616,Z 985.245,A -85,B 0,C 180,E1 10715.231,E2 10715.231} C_VEL
LIN {X 0,Y 208.76,Z 986.048,A -85,B 0,C 180,E1 10710.829,E2 10710.829} C_VEL
LIN {X 0,Y 208.684,Z 985.875,A -85,B 0,C 180,E1 10706.71,E2 10706.71} C_VEL
LIN {X 0,Y 208.478,Z 984.532,A -85,B 0,C 180,E1 10701.734,E2 10701.734} C_VEL
LIN {X 0,Y 208.664,Z 981.623,A -85,B 0,C 180,E1 10696.427,E2 10696.427} C_VEL
LIN {X 0,Y 209.95,Z 976.9,A -85,B 0,C 180,E1 10690.534,E2 10690.534} C_VEL
LIN {X 0,Y 212.741,Z 970.419,A -85,B 0,C 180,E1 10684.686,E2 10684.686} C_VEL
LIN {X 0,Y 217.258,Z 962.085,A -85,B 0,C 180,E1 10678.981,E2 10678.981} C_VEL
LIN {X 0,Y 223.586,Z 951.849,A -85,B 0,C 180,E1 10673.512,E2 10673.512} C_VEL
LIN {X 0,Y 230.857,Z 940.792,A -85,B 0,C 180,E1 10668.837,E2 10668.837} C_VEL
LIN {X 0,Y 239.519,Z 927.666,A -85,B 0,C 180,E1 10664.462,E2 10664.462} C_VEL
LIN {X 0,Y 248.361,Z 913.931,A -85,B 0,C 180,E1 10660.822,E2 10660.822} C_VEL
LIN {X 0,Y 258.169,Z 898.07,A -85,B 0,C 180,E1 10657.455,E2 10657.455} C_VEL
LIN {X 0,Y 267.875,Z 881.242,A -85,B 0,C 180,E1 10654.622,E2 10654.622} C_VEL
LIN {X 0,Y 277.227,Z 863.426,A -85,B 0,C 180,E1 10652.261,E2 10652.261} C_VEL
LIN {X 0,Y 285.995,Z 844.748,A -85,B 0,C 180,E1 10650.296,E2 10650.296} C_VEL
LIN {X 0,Y 294.031,Z 825.43,A -85,B 0,C 180,E1 10648.69,E2 10648.69} C_VEL
LIN {X 0,Y 300.817,Z 806.47,A -85,B 0,C 180,E1 10647.457,E2 10647.457} C_VEL
LIN {X 0,Y 306.614,Z 786.944,A -85,B 0,C 180,E1 10646.487,E2 10646.487} C_VEL
LIN {X 0,Y 311.869,Z 764.871,A -85,B 0,C 180,E1 10645.666,E2 10645.666} C_VEL
LIN {X 0,Y 315.548,Z 743.041,A -85,B 0,C 180,E1 10645.05,E2 10645.05} C_VEL
LIN {X 0,Y 331.995,Z 580.62,A -85,B 0,C 180,E1 10641.579,E2 10641.579} C_VEL
LIN {X 0,Y 329.36,Z 574.157,A -85,B 0,C 180,E1 10639.047,E2 10639.047} C_VEL
LIN {X 0,Y 327.58,Z 570.079,A -85,B 0,C 180,E1 10636.764,E2 10636.764} C_VEL
LIN {X 0,Y 326.776,Z 568.476,A -85,B 0,C 180,E1 10635.438,E2 10635.438} C_VEL
LIN {X 0,Y 325.859,Z 565.801,A -85,B 0,C 180,E1 10632.583,E2 10632.583} C_VEL
LIN {X 0,Y 325.808,Z 565.928,A -85,B 0,C 180,E1 10629.182,E2 10629.182} C_VEL
LIN {X 0,Y 327.113,Z 569.675,A -85,B 0,C 180,E1 10625.525,E2 10625.525} C_VEL
LIN {X 0,Y 328.784,Z 573.81,A -85,B 0,C 180,E1 10623.137,E2 10623.137} C_VEL
LIN {X 0,Y 331.228,Z 580.071,A -85,B 0,C 180,E1 10620.605,E2 10620.605} C_VEL
LIN {X 0,Y 314.331,Z 734.438,A -85,B 0,C 180,E1 10617.256,E2 10617.256} C_VEL
LIN {X 0,Y 310.64,Z 755.311,A -85,B 0,C 180,E1 10616.564,E2 10616.564} C_VEL
LIN {X 0,Y 305.809,Z 775.483,A -85,B 0,C 180,E1 10615.646,E2 10615.646} C_VEL
LIN {X 0,Y 299.795,Z 795.507,A -85,B 0,C 180,E1 10614.449,E2 10614.449} C_VEL
LIN {X 0,Y 293.09,Z 814.021,A -85,B 0,C 180,E1 10613.037,E2 10613.037} C_VEL
LIN {X 0,Y 285.235,Z 832.285,A -85,B 0,C 180,E1 10611.269,E2 10611.269} C_VEL
LIN {X 0,Y 276.72,Z 849.606,A -85,B 0,C 180,E1 10609.17,E2 10609.17} C_VEL
LIN {X 0,Y 267.388,Z 866.44,A -85,B 0,C 180,E1 10606.594,E2 10606.594} C_VEL
LIN {X 0,Y 258.277,Z 881.335,A -85,B 0,C 180,E1 10603.731,E2 10603.731} C_VEL
LIN {X 0,Y 249.281,Z 894.851,A -85,B 0,C 180,E1 10600.469,E2 10600.469} C_VEL
LIN {X 0,Y 240.226,Z 907.482,A -85,B 0,C 180,E1 10596.583,E2 10596.583} C_VEL
LIN {X 0,Y 232.28,Z 917.948,A -85,B 0,C 180,E1 10592.451,E2 10592.451} C_VEL
LIN {X 0,Y 224.908,Z 927.439,A -85,B 0,C 180,E1 10587.624,E2 10587.624} C_VEL
LIN {X 0,Y 219.04,Z 934.96,A -85,B 0,C 180,E1 10582.574,E2 10582.574} C_VEL
LIN {X 0,Y 214.502,Z 940.97,A -85,B 0,C 180,E1 10577.112,E2 10577.112} C_VEL
LIN {X 0,Y 211.31,Z 945.446,A -85,B 0,C 180,E1 10571.116,E2 10571.116} C_VEL
LIN {X 0,Y 209.713,Z 947.844,A -85,B 0,C 180,E1 10565.559,E2 10565.559} C_VEL
LIN {X 0,Y 209.051,Z 948.785,A -85,B 0,C 180,E1 10560.036,E2 10560.036} C_VEL
LIN {X 0,Y 208.957,Z 948.424,A -85,B 0,C 180,E1 10554.895,E2 10554.895} C_VEL
LIN {X 0,Y 209.349,Z 946.582,A -85,B 0,C 180,E1 10549.525,E2 10549.525} C_VEL
LIN {X 0,Y 210.522,Z 943.235,A -85,B 0,C 180,E1 10544.011,E2 10544.011} C_VEL
LIN {X 0,Y 212.759,Z 938.41,A -85,B 0,C 180,E1 10538.643,E2 10538.643} C_VEL
LIN {X 0,Y 216.428,Z 931.601,A -85,B 0,C 180,E1 10533.172,E2 10533.172} C_VEL
LIN {X 0,Y 221.215,Z 923.316,A -85,B 0,C 180,E1 10528.181,E2 10528.181} C_VEL
LIN {X 0,Y 227.269,Z 913.178,A -85,B 0,C 180,E1 10523.427,E2 10523.427} C_VEL
LIN {X 0,Y 234.15,Z 901.605,A -85,B 0,C 180,E1 10519.159,E2 10519.159} C_VEL
LIN {X 0,Y 241.557,Z 888.697,A -85,B 0,C 180,E1 10515.37,E2 10515.37} C_VEL
LIN {X 0,Y 249.336,Z 874.382,A -85,B 0,C 180,E1 10512.01,E2 10512.01} C_VEL
LIN {X 0,Y 257.504,Z 857.971,A -85,B 0,C 180,E1 10508.947,E2 10508.947} C_VEL
LIN {X 0,Y 265.382,Z 840.375,A -85,B 0,C 180,E1 10506.339,E2 10506.339} C_VEL
LIN {X 0,Y 272.499,Z 822.459,A -85,B 0,C 180,E1 10504.223,E2 10504.223} C_VEL
LIN {X 0,Y 278.946,Z 803.78,A -85,B 0,C 180,E1 10502.455,E2 10502.455} C_VEL
LIN {X 0,Y 284.769,Z 783.792,A -85,B 0,C 180,E1 10500.96,E2 10500.96} C_VEL
LIN {X 0,Y 289.646,Z 763.171,A -85,B 0,C 180,E1 10499.775,E2 10499.775} C_VEL
LIN {X 0,Y 293.616,Z 741.08,A -85,B 0,C 180,E1 10498.846,E2 10498.846} C_VEL
LIN {X 0,Y 296.3,Z 718.523,A -85,B 0,C 180,E1 10498.204,E2 10498.204} C_VEL
LIN {X 0,Y 309.144,Z 568.055,A -85,B 0,C 180,E1 10494.867,E2 10494.867} C_VEL
LIN {X 0,Y 302.82,Z 556.59,A -85,B 0,C 180,E1 10492.106,E2 10492.106} C_VEL
LIN {X 0,Y 296.323,Z 545.682,A -85,B 0,C 180,E1 10488.951,E2 10488.951} C_VEL
LIN {X 0,Y 290.197,Z 536.06,A -85,B 0,C 180,E1 10485.575,E2 10485.575} C_VEL
LIN {X 0,Y 285.487,Z 528.929,A -85,B 0,C 180,E1 10482.606,E2 10482.606} C_VEL
LIN {X 0,Y 282.206,Z 524.275,A -85,B 0,C 180,E1 10480.286,E2 10480.286} C_VEL
LIN {X 0,Y 279.093,Z 519.792,A -85,B 0,C 180,E1 10477.779,E2 10477.779} C_VEL
LIN {X 0,Y 275.572,Z 514.834,A -85,B 0,C 180,E1 10474.474,E2 10474.474} C_VEL
LIN {X 0,Y 272.004,Z 509.962,A -85,B 0,C 180,E1 10470.239,E2 10470.239} C_VEL
LIN {X 0,Y 268.345,Z 505.033,A -85,B 0,C 180,E1 10463.264,E2 10463.264} C_VEL
LIN {X 0,Y 267.731,Z 504.485,A -85,B 0,C 180,E1 10461.177,E2 10461.177} C_VEL
LIN {X 0,Y 267.282,Z 505.171,A -85,B 0,C 180,E1 10459.526,E2 10459.526} C_VEL
LIN {X 0,Y 266.368,Z 511.61,A -85,B 0,C 180,E1 10454.788,E2 10454.788} C_VEL
LIN {X 0,Y 266.449,Z 512.199,A -85,B 0,C 180,E1 10453.713,E2 10453.713} C_VEL
LIN {X 0,Y 267.642,Z 513.478,A -85,B 0,C 180,E1 10449.495,E2 10449.495} C_VEL
LIN {X 0,Y 271.581,Z 518.786,A -85,B 0,C 180,E1 10442.638,E2 10442.638} C_VEL
LIN {X 0,Y 275.501,Z 524.22,A -85,B 0,C 180,E1 10438.233,E2 10438.233} C_VEL
LIN {X 0,Y 279.396,Z 529.736,A -85,B 0,C 180,E1 10434.765,E2 10434.765} C_VEL
LIN {X 0,Y 283.489,Z 535.618,A -85,B 0,C 180,E1 10431.686,E2 10431.686} C_VEL
LIN {X 0,Y 288.773,Z 543.506,A -85,B 0,C 180,E1 10428.264,E2 10428.264} C_VEL
LIN {X 0,Y 295.101,Z 553.345,A -85,B 0,C 180,E1 10424.727,E2 10424.727} C_VEL
LIN {X 0,Y 301.479,Z 563.943,A -85,B 0,C 180,E1 10421.586,E2 10421.586} C_VEL
LIN {X 0,Y 308.463,Z 576.225,A -85,B 0,C 180,E1 10418.514,E2 10418.514} C_VEL
LIN {X 0,Y 309.179,Z 577.902,A -85,B 0,C 180,E1 10418.2,E2 10418.2} C_VEL
LIN {X 0,Y 295.041,Z 748.003,A -85,B 0,C 180,E1 10414.534,E2 10414.534} C_VEL
LIN {X 0,Y 291.607,Z 770.198,A -85,B 0,C 180,E1 10413.849,E2 10413.849} C_VEL
LIN {X 0,Y 287.039,Z 791.039,A -85,B 0,C 180,E1 10412.988,E2 10412.988} C_VEL
LIN {X 0,Y 281.318,Z 811.957,A -85,B 0,C 180,E1 10411.822,E2 10411.822} C_VEL
LIN {X 0,Y 274.868,Z 831.623,A -85,B 0,C 180,E1 10410.393,E2 10410.393} C_VEL
LIN {X 0,Y 267.242,Z 851.351,A -85,B 0,C 180,E1 10408.55,E2 10408.55} C_VEL
LIN {X 0,Y 259.29,Z 869.526,A -85,B 0,C 180,E1 10406.406,E2 10406.406} C_VEL
LIN {X 0,Y 250.866,Z 886.896,A -85,B 0,C 180,E1 10403.853,E2 10403.853} C_VEL
LIN {X 0,Y 242.209,Z 903.255,A -85,B 0,C 180,E1 10400.833,E2 10400.833} C_VEL
LIN {X 0,Y 233.729,Z 918.121,A -85,B 0,C 180,E1 10397.38,E2 10397.38} C_VEL
LIN {X 0,Y 225.561,Z 931.946,A -85,B 0,C 180,E1 10393.368,E2 10393.368} C_VEL
LIN {X 0,Y 218.191,Z 944.268,A -85,B 0,C 180,E1 10388.894,E2 10388.894} C_VEL
LIN {X 0,Y 211.665,Z 955.414,A -85,B 0,C 180,E1 10383.76,E2 10383.76} C_VEL
LIN {X 0,Y 206.62,Z 964.68,A -85,B 0,C 180,E1 10378.273,E2 10378.273} C_VEL
LIN {X 0,Y 202.999,Z 972.616,A -85,B 0,C 180,E1 10372.185,E2 10372.185} C_VEL
LIN {X 0,Y 201.095,Z 978.475,A -85,B 0,C 180,E1 10366.173,E2 10366.173} C_VEL
LIN {X 0,Y 200.536,Z 982.241,A -85,B 0,C 180,E1 10360.637,E2 10360.637} C_VEL
LIN {X 0,Y 200.648,Z 984.564,A -85,B 0,C 180,E1 10355.152,E2 10355.152} C_VEL
LIN {X 0,Y 200.795,Z 985.334,A -85,B 0,C 180,E1 10350.577,E2 10350.577} C_VEL
LIN {X 0,Y 200.692,Z 985.123,A -85,B 0,C 180,E1 10346.293,E2 10346.293} C_VEL
LIN {X 0,Y 200.478,Z 983.717,A -85,B 0,C 180,E1 10341.112,E2 10341.112} C_VEL
LIN {X 0,Y 200.771,Z 980.76,A -85,B 0,C 180,E1 10335.588,E2 10335.588} C_VEL
LIN {X 0,Y 202.394,Z 975.694,A -85,B 0,C 180,E1 10329.171,E2 10329.171} C_VEL
LIN {X 0,Y 205.643,Z 969.129,A -85,B 0,C 180,E1 10323.124,E2 10323.124} C_VEL
LIN {X 0,Y 210.724,Z 960.651,A -85,B 0,C 180,E1 10317.262,E2 10317.262} C_VEL
LIN {X 0,Y 217.679,Z 950.251,A -85,B 0,C 180,E1 10311.686,E2 10311.686} C_VEL
LIN {X 0,Y 225.995,Z 938.395,A -85,B 0,C 180,E1 10306.714,E2 10306.714} C_VEL
LIN {X 0,Y 235.341,Z 925.087,A -85,B 0,C 180,E1 10302.342,E2 10302.342} C_VEL
LIN {X 0,Y 245.364,Z 910.225,A -85,B 0,C 180,E1 10298.529,E2 10298.529} C_VEL
LIN {X 0,Y 255.471,Z 894.349,A -85,B 0,C 180,E1 10295.322,E2 10295.322} C_VEL
LIN {X 0,Y 265.733,Z 876.946,A -85,B 0,C 180,E1 10292.551,E2 10292.551} C_VEL
LIN {X 0,Y 275.481,Z 858.75,A -85,B 0,C 180,E1 10290.264,E2 10290.264} C_VEL
LIN {X 0,Y 284.25,Z 840.336,A -85,B 0,C 180,E1 10288.444,E2 10288.444} C_VEL
LIN {X 0,Y 292.568,Z 820.185,A -85,B 0,C 180,E1 10286.89,E2 10286.89} C_VEL
LIN {X 0,Y 299.979,Z 799.018,A -85,B 0,C 180,E1 10285.644,E2 10285.644} C_VEL
LIN {X 0,Y 306.016,Z 777.891,A -85,B 0,C 180,E1 10284.722,E2 10284.722} C_VEL
LIN {X 0,Y 310.794,Z 755.977,A -85,B 0,C 180,E1 10284.012,E2 10284.012} C_VEL
LIN {X 0,Y 314.026,Z 733.303,A -85,B 0,C 180,E1 10283.449,E2 10283.449} C_VEL
LIN {X 0,Y 329.42,Z 585.76,A -85,B 0,C 180,E1 10280.317,E2 10280.317} C_VEL
LIN {X 0,Y 327.261,Z 580.059,A -85,B 0,C 180,E1 10277.881,E2 10277.881} C_VEL
LIN {X 0,Y 325.818,Z 576.706,A -85,B 0,C 180,E1 10275.667,E2 10275.667} C_VEL
LIN {X 0,Y 324.753,Z 573.708,A -85,B 0,C 180,E1 10272.445,E2 10272.445} C_VEL
LIN {X 0,Y 324.686,Z 573.76,A -85,B 0,C 180,E1 10269.393,E2 10269.393} C_VEL
LIN {X 0,Y 325.884,Z 577.562,A -85,B 0,C 180,E1 10265.722,E2 10265.722} C_VEL
LIN {X 0,Y 327.391,Z 581.582,A -85,B 0,C 180,E1 10263.414,E2 10263.414} C_VEL
LIN {X 0,Y 328.725,Z 585.478,A -85,B 0,C 180,E1 10261.841,E2 10261.841} C_VEL
LIN {X 0,Y 311.809,Z 734.899,A -85,B 0,C 180,E1 10258.644,E2 10258.644} C_VEL
LIN {X 0,Y 307.948,Z 756.083,A -85,B 0,C 180,E1 10257.953,E2 10257.953} C_VEL
LIN {X 0,Y 303.073,Z 775.896,A -85,B 0,C 180,E1 10257.068,E2 10257.068} C_VEL
LIN {X 0,Y 297.147,Z 795.112,A -85,B 0,C 180,E1 10255.947,E2 10255.947} C_VEL
LIN {X 0,Y 289.96,Z 814.347,A -85,B 0,C 180,E1 10254.509,E2 10254.509} C_VEL
LIN {X 0,Y 282.134,Z 832.033,A -85,B 0,C 180,E1 10252.833,E2 10252.833} C_VEL
LIN {X 0,Y 273.449,Z 849.172,A -85,B 0,C 180,E1 10250.801,E2 10250.801} C_VEL
LIN {X 0,Y 263.913,Z 865.889,A -85,B 0,C 180,E1 10248.305,E2 10248.305} C_VEL
LIN {X 0,Y 254.485,Z 880.778,A -85,B 0,C 180,E1 10245.506,E2 10245.506} C_VEL
LIN {X 0,Y 244.368,Z 895.324,A -85,B 0,C 180,E1 10242.023,E2 10242.023} C_VEL
LIN {X 0,Y 234.843,Z 907.919,A -85,B 0,C 180,E1 10238.129,E2 10238.129} C_VEL
LIN {X 0,Y 226.064,Z 918.886,A -85,B 0,C 180,E1 10233.749,E2 10233.749} C_VEL
LIN {X 0,Y 218.238,Z 928.315,A -85,B 0,C 180,E1 10228.82,E2 10228.82} C_VEL
LIN {X 0,Y 211.713,Z 936.103,A -85,B 0,C 180,E1 10223.392,E2 10223.392} C_VEL
LIN {X 0,Y 206.934,Z 941.933,A -85,B 0,C 180,E1 10217.807,E2 10217.807} C_VEL
LIN {X 0,Y 203.637,Z 946.172,A -85,B 0,C 180,E1 10211.885,E2 10211.885} C_VEL
LIN {X 0,Y 201.854,Z 948.572,A -85,B 0,C 180,E1 10206.109,E2 10206.109} C_VEL
LIN {X 0,Y 201.109,Z 949.511,A -85,B 0,C 180,E1 10200.464,E2 10200.464} C_VEL
LIN {X 0,Y 200.982,Z 949.17,A -85,B 0,C 180,E1 10195.117,E2 10195.117} C_VEL
LIN {X 0,Y 201.347,Z 947.45,A -85,B 0,C 180,E1 10189.728,E2 10189.728} C_VEL
LIN {X 0,Y 202.545,Z 944.21,A -85,B 0,C 180,E1 10183.991,E2 10183.991} C_VEL
LIN {X 0,Y 204.854,Z 939.493,A -85,B 0,C 180,E1 10178.414,E2 10178.414} C_VEL
LIN {X 0,Y 208.657,Z 932.742,A -85,B 0,C 180,E1 10172.741,E2 10172.741} C_VEL
LIN {X 0,Y 213.637,Z 924.582,A -85,B 0,C 180,E1 10167.58,E2 10167.58} C_VEL
LIN {X 0,Y 219.928,Z 914.573,A -85,B 0,C 180,E1 10162.681,E2 10162.681} C_VEL
LIN {X 0,Y 227.056,Z 903.16,A -85,B 0,C 180,E1 10158.308,E2 10158.308} C_VEL
LIN {X 0,Y 234.741,Z 890.392,A -85,B 0,C 180,E1 10154.429,E2 10154.429} C_VEL
LIN {X 0,Y 242.77,Z 876.186,A -85,B 0,C 180,E1 10151.008,E2 10151.008} C_VEL
LIN {X 0,Y 250.911,Z 860.52,A -85,B 0,C 180,E1 10147.997,E2 10147.997} C_VEL
LIN {X 0,Y 258.707,Z 843.972,A -85,B 0,C 180,E1 10145.447,E2 10145.447} C_VEL
LIN {X 0,Y 266.317,Z 825.874,A -85,B 0,C 180,E1 10143.218,E2 10143.218} C_VEL
LIN {X 0,Y 272.943,Z 807.84,A -85,B 0,C 180,E1 10141.438,E2 10141.438} C_VEL
LIN {X 0,Y 279.093,Z 788.029,A -85,B 0,C 180,E1 10139.893,E2 10139.893} C_VEL
LIN {X 0,Y 284.195,Z 767.753,A -85,B 0,C 180,E1 10138.676,E2 10138.676} C_VEL
LIN {X 0,Y 288.336,Z 746.574,A -85,B 0,C 180,E1 10137.726,E2 10137.726} C_VEL
LIN {X 0,Y 291.4,Z 724.221,A -85,B 0,C 180,E1 10137.028,E2 10137.028} C_VEL
LIN {X 0,Y 304.884,Z 572.139,A -85,B 0,C 180,E1 10133.661,E2 10133.661} C_VEL
LIN {X 0,Y 297.71,Z 559.17,A -85,B 0,C 180,E1 10130.323,E2 10130.323} C_VEL
LIN {X 0,Y 291.835,Z 549.252,A -85,B 0,C 180,E1 10127.239,E2 10127.239} C_VEL
LIN {X 0,Y 285.411,Z 539.096,A -85,B 0,C 180,E1 10123.365,E2 10123.365} C_VEL
LIN {X 0,Y 280.657,Z 532.044,A -85,B 0,C 180,E1 10120.004,E2 10120.004} C_VEL
LIN {X 0,Y 277.346,Z 527.243,A -85,B 0,C 180,E1 10117.277,E2 10117.277} C_VEL
LIN {X 0,Y 274.068,Z 522.486,A -85,B 0,C 180,E1 10114.086,E2 10114.086} C_VEL
LIN {X 0,Y 270.668,Z 517.717,A -85,B 0,C 180,E1 10109.914,E2 10109.914} C_VEL
LIN {X 0,Y 267.223,Z 512.933,A -85,B 0,C 180,E1 10103.134,E2 10103.134} C_VEL
LIN {X 0,Y 266.194,Z 512.016,A -85,B 0,C 180,E1 10097.713,E2 10097.713} C_VEL
LIN {X 0,Y 266.449,Z 512.199,A -85,B 0,C 180,E1 10093.713,E2 10093.713} C_VEL
LIN {X 0,Y 266.642,Z 513.458,A -85,B 0,C 180,E1 10092.188,E2 10092.188} C_VEL
LIN {X 0,Y 266.893,Z 517.972,A -85,B 0,C 180,E1 10089.853,E2 10089.853} C_VEL
LIN {X 0,Y 267.517,Z 522.761,A -85,B 0,C 180,E1 10087.399,E2 10087.399} C_VEL
LIN {X 0,Y 267.942,Z 523.757,A -85,B 0,C 180,E1 10086.466,E2 10086.466} C_VEL
LIN {X 0,Y 270.312,Z 526.669,A -85,B 0,C 180,E1 10082.864,E2 10082.864} C_VEL
LIN {X 0,Y 273.963,Z 531.832,A -85,B 0,C 180,E1 10078.641,E2 10078.641} C_VEL
LIN {X 0,Y 277.774,Z 537.38,A -85,B 0,C 180,E1 10075.148,E2 10075.148} C_VEL
LIN {X 0,Y 281.801,Z 543.285,A -85,B 0,C 180,E1 10072.047,E2 10072.047} C_VEL
LIN {X 0,Y 286.848,Z 551.027,A -85,B 0,C 180,E1 10068.693,E2 10068.693} C_VEL
LIN {X 0,Y 293.601,Z 561.745,A -85,B 0,C 180,E1 10064.849,E2 10064.849} C_VEL
LIN {X 0,Y 300.781,Z 574.16,A -85,B 0,C 180,E1 10061.29,E2 10061.29} C_VEL
LIN {X 0,Y 304.905,Z 581.912,A -85,B 0,C 180,E1 10059.418,E2 10059.418} C_VEL
LIN {X 0,Y 290.696,Z 747.725,A -85,B 0,C 180,E1 10055.853,E2 10055.853} C_VEL
LIN {X 0,Y 287.176,Z 769.954,A -85,B 0,C 180,E1 10055.172,E2 10055.172} C_VEL
LIN {X 0,Y 282.409,Z 791.136,A -85,B 0,C 180,E1 10054.302,E2 10054.302} C_VEL
LIN {X 0,Y 276.42,Z 812.36,A -85,B 0,C 180,E1 10053.119,E2 10053.119} C_VEL
LIN {X 0,Y 269.697,Z 832.217,A -85,B 0,C 180,E1 10051.671,E2 10051.671} C_VEL
LIN {X 0,Y 261.582,Z 852.478,A -85,B 0,C 180,E1 10049.758,E2 10049.758} C_VEL
LIN {X 0,Y 253.415,Z 870.358,A -85,B 0,C 180,E1 10047.608,E2 10047.608} C_VEL
LIN {X 0,Y 244.379,Z 888.177,A -85,B 0,C 180,E1 10044.92,E2 10044.92} C_VEL
LIN {X 0,Y 235.768,Z 903.822,A -85,B 0,C 180,E1 10041.962,E2 10041.962} C_VEL
LIN {X 0,Y 226.536,Z 919.375,A -85,B 0,C 180,E1 10038.244,E2 10038.244} C_VEL
LIN {X 0,Y 218.175,Z 932.818,A -85,B 0,C 180,E1 10034.16,E2 10034.16} C_VEL
LIN {X 0,Y 210.152,Z 945.54,A -85,B 0,C 180,E1 10029.262,E2 10029.262} C_VEL
LIN {X 0,Y 203.627,Z 956.184,A -85,B 0,C 180,E1 10024.046,E2 10024.046} C_VEL
LIN {X 0,Y 198.446,Z 965.349,A -85,B 0,C 180,E1 10018.275,E2 10018.275} C_VEL
LIN {X 0,Y 194.991,Z 972.56,A -85,B 0,C 180,E1 10012.306,E2 10012.306} C_VEL
LIN {X 0,Y 193.055,Z 978.297,A -85,B 0,C 180,E1 10005.938,E2 10005.938} C_VEL
LIN {X 0,Y 192.539,Z 981.935,A -85,B 0,C 180,E1 10000.176,E2 10000.176} C_VEL
LIN {X 0,Y 192.691,Z 983.949,A -85,B 0,C 180,E1 9994.769,E2 9994.769} C_VEL
